(*Gestion des fronts demandes*)
FM_On.CLK	:=	CO_Etat;
FM_On();
IF FM_On.Q THEN
	VAR_Mem_CO_On	:=	TRUE;
END_IF
FD_Off.CLK	:=	CO_Etat;
FD_Off();
IF FD_Off.Q THEN
	VAR_Mem_CO_Off	:=	TRUE;
END_IF
FM_Regen.CLK	:=	CO_Regen;
FM_Regen();
IF FM_Regen.Q THEN
	VAR_Mem_CO_Regen	:=	TRUE;
	VAR_Mem_etape_Regen := TRUE;
END_IF
FM_states_regen.CLK	:=	CO_states_regen;
FM_states_regen();
IF FM_states_regen.Q THEN
	VAR_Mem_etape_Regen := TRUE;
END_IF
FM_StopRegen.CLK	:=	CO_StopRegen;
FM_StopRegen();
IF FM_StopRegen.Q THEN
	VAR_Mem_CO_StopRegen	:=	TRUE;
	VAR_Mem_etape_Regen := FALSE;
END_IF
FM_Param.CLK	:=	CO_Param_ParDefaut;
FM_Param();
IF FM_Param.Q THEN
	VAR_Mem_CO_Param_ParDefaut	:=	TRUE;
END_IF           
FM_Ecriture.CLK	:=	CO_Ecriture;
FM_Ecriture();
IF FM_Ecriture.Q THEN
	VAR_Mem_CO_Ecriture	:=	TRUE;
END_IF
FM_Lecture.CLK	:=	CO_Lecture;
FM_Lecture();
IF FM_Lecture.Q THEN
	VAR_Mem_CO_Lecture	:=	TRUE;
END_IF
FM_RoughValveOn.CLK	:=	CO_RoughValve;
FM_RoughValveOn();
IF FM_RoughValveOn.Q THEN
	VAR_Mem_CO_RoughValve_On	:=	TRUE;
END_IF
FM_PurgeValveOn.CLK	:=	CO_PurgeValve;
FM_PurgeValveOn();
IF FM_PurgeValveOn.Q THEN
	VAR_Mem_CO_PurgeValve_On	:=	TRUE;
END_IF
FM_RoughValveOff.CLK	:=	CO_RoughValve;
FM_RoughValveOff();
IF FM_RoughValveOff.Q THEN
	VAR_Mem_CO_RoughValve_Off	:=	TRUE;
END_IF
FM_PurgeValveOff.CLK	:=	CO_PurgeValve;
FM_PurgeValveOff();
IF FM_PurgeValveOff.Q THEN
	VAR_Mem_CO_PurgeValve_Off	:=	TRUE;
END_IF

FM_pump_TC_ON.CLK	:=	CO_PumpTc;
FM_pump_TC_ON();
IF FM_pump_TC_ON.Q THEN
	VAR_Mem_CO_PumpTC_on	:=	TRUE;
END_IF
FM_pump_TC_OFF.CLK	:=	CO_PumpTc;
FM_pump_TC_OFF();
IF FM_pump_TC_OFF.Q THEN
	VAR_Mem_CO_PumpTC_off	:=	TRUE;
END_IF



FM_InfoPompe.CLK	:=	CO_InfoPompe;
FM_InfoPompe();
IF FM_InfoPompe.Q THEN
	VAR_Mem_CO_Info_Pompe	:=	TRUE;
END_IF
FM_LectureRelay.CLK := CO_Lecture_Relay;
FM_LectureRelay();
IF FM_LectureRelay.Q THEN
	VAR_Mem_CO_Lecture_Relay:=TRUE;
END_IF
FM_EnvoieParamRelay.CLK	:=	CO_Envoie_Param_Relay;
FM_EnvoieParamRelay();
IF FM_EnvoieParamRelay.Q THEN
	VAR_Mem_CO_Envoie_Param_Relay	:=	TRUE;
END_IF
FM_ParamUsineRelay.CLK	:=	CO_Param_usine_Relay;
FM_ParamUsineRelay();
IF FM_ParamUsineRelay.Q THEN
	VAR_Mem_CO_Param_usine_Relay	:=	TRUE;
END_IF

IF NOT CO_Etat THEN
	STATE_Pompe:= FALSE;
END_IF

A_error:= OUT_Send_Data.Error;


(*RESET ou DESACTIVATION Driver*)
IF RESET OR OFF THEN
	VAR_Cadence                 := 0;
	STATE_Temperature[0]		:=	0;
	STATE_Temperature[1]		:=	0;
	STATE_Pressure        		:=  0;
	REGEN_ERROR                 := '';
	Reponse_ModeManu            := '';
	STEP_Regen                  := '';
	STATE_ROR_nb                := 0;
	LAST_ROR_Value              := 0;
	STATE_Rough_valve           := FALSE;
	STATE_Purge_valve           := FALSE;
	STEP_REGEN_ID               := 1000;
	VAR_Affichage               := '';
	Pump_Serial_Number_affiche	:= '';
	Number_Of_Complete_Regen    := 0;
	Time_Since_Last_Regen       := 0;
	SoftwareRevisionLevel       := '';
	ElaspedTime                 := 0;
	STATE_Tps_restant           := 0;
	VAR_Mem_CO_Ecriture   		:= FALSE;
	VAR_Mem_CO_Param_ParDefaut  := FALSE;
	VAR_Mem_CO_On				:= FALSE;
	VAR_Mem_CO_Off		  		:= TRUE ;
	VAR_Mem_CO_Regen	 		:= FALSE;
	VAR_Mem_CO_StopRegen 		:= TRUE ;
	VAR_Mem_CO_PurgeValve_off   := TRUE ;
	VAR_Mem_CO_PurgeValve_on    := FALSE;
	VAR_Mem_CO_RoughValve_off   := TRUE ;
	VAR_Mem_CO_RoughValve_on    := FALSE;
	VAR_Mem_CO_Info_Pompe		:= FALSE;
	RETURN;
END_IF



TIMER_Demarrage.IN 	:= 	NOT IN_Receive_Data.Busy AND NOT OUT_Send_Data.Busy AND NOT VAR_ReceptionOk;
TIMER_Demarrage.PT	:=	T#5S;
TIMER_Demarrage();
IF TIMER_Demarrage.Q  THEN
	VAR_ReceptionOk	:=	TRUE;
	VAR_Cadence 	:= 	1;
END_IF

(*Cadencement des trames*)
TIMER_Cadence(IN:=VAR_ReceptionOk, PT:=T#500MS);
VAR_Mem_Cadence	:=	VAR_Cadence;



(*GESTION ENVOI*)
IF TIMER_Cadence.Q AND NOT OUT_Send_Data.Busy AND NOT CO_ModeManu THEN
	VAR_STR2 := CHR(36);	(*$ = hex 24 = dec 36*)

	(* Remplissage trame : $ + code + checksum + 0D*)
	CASE VAR_Cadence OF

			1: 	(* Demande état on/off pompe*)
				VAR_BuffString		:= 	'';
				VAR_BuffString		:=	VAR_STR2;
				VAR_BuffString		:=	CONCAT(VAR_BuffString, 'A?');
				VAR_BuffString		:=	CONCAT(VAR_BuffString,CHECKSUM(VAR_BuffString,TRUE));
				VAR_BuffString		:=	CONCAT(VAR_BuffString,'$0D');
				OUT_Send_Data.SendString		:=	VAR_BuffString;

			2: 	(* Demande état regen pompe*)
				VAR_BuffString		:= 	'';
				VAR_BuffString		:=	VAR_STR2;
				VAR_BuffString		:=	CONCAT(VAR_BuffString, 'O');
				VAR_BuffString		:=	CONCAT(VAR_BuffString,CHECKSUM(VAR_BuffString,TRUE));
				VAR_BuffString		:=	CONCAT(VAR_BuffString,'$0D');
				OUT_Send_Data.SendString		:=	VAR_BuffString;
				
			3:	(* Demande erreur regen *)
				VAR_BuffString		:= 	'';
				VAR_BuffString		:=	VAR_STR2;
				VAR_BuffString		:=	CONCAT(VAR_BuffString, 'e');
				VAR_BuffString		:=	CONCAT(VAR_BuffString,CHECKSUM(VAR_BuffString,TRUE));
				VAR_BuffString		:=	CONCAT(VAR_BuffString,'$0D');
				OUT_Send_Data.SendString		:=	VAR_BuffString;
				
			4: 	(* Demande etat rough valve *)
				VAR_BuffString		:= 	'';
				VAR_BuffString		:=	VAR_STR2;
				VAR_BuffString		:=	CONCAT(VAR_BuffString, 'D?');
				VAR_BuffString		:=	CONCAT(VAR_BuffString,CHECKSUM(VAR_BuffString,TRUE));
				VAR_BuffString		:=	CONCAT(VAR_BuffString,'$0D');
				OUT_Send_Data.SendString	:=	VAR_BuffString;
				
			5: 	(* Demande etat purge valve *)
				VAR_BuffString		:= 	'';
				VAR_BuffString		:=	VAR_STR2;
				VAR_BuffString		:=	CONCAT(VAR_BuffString, 'E?');
				VAR_BuffString		:=	CONCAT(VAR_BuffString,CHECKSUM(VAR_BuffString,TRUE));
				VAR_BuffString		:=	CONCAT(VAR_BuffString,'$0D');
				OUT_Send_Data.SendString	:=	VAR_BuffString;
		
			
			6: 	(* Demande température étage 1*)
				VAR_BuffString		:= 	'';
				VAR_BuffString		:=	VAR_STR2;
				VAR_BuffString		:=	CONCAT(VAR_BuffString, 'J');
				VAR_BuffString		:=	CONCAT(VAR_BuffString,CHECKSUM(VAR_BuffString,TRUE));
				VAR_BuffString		:=	CONCAT(VAR_BuffString,CHR(13));
				VAR_TrameRetour     :=  VAR_BuffString;
				OUT_Send_Data.SendString	:=	VAR_BuffString;
				
			7: 	(* Demande température étage 2*)
				VAR_BuffString		:= 	'';
				VAR_BuffString		:=	VAR_STR2;
				VAR_BuffString		:=	CONCAT(VAR_BuffString, 'K');
				VAR_BuffString		:=	CONCAT(VAR_BuffString,CHECKSUM(VAR_BuffString,TRUE));
				VAR_BuffString		:=	CONCAT(VAR_BuffString,'$0D');
				OUT_Send_Data.SendString		:=	VAR_BuffString;
				
			8: 	(* Demande pression *)
				VAR_BuffString		:= 	'';
				VAR_BuffString		:=	VAR_STR2;
				VAR_BuffString		:=	CONCAT(VAR_BuffString, 'L');
				VAR_BuffString		:=	CONCAT(VAR_BuffString,CHECKSUM(VAR_BuffString,TRUE));
				VAR_BuffString		:=	CONCAT(VAR_BuffString,'$0D');
				OUT_Send_Data.SendString	:=	VAR_BuffString;
				
			9: 	(* Demande etat pump TC *)
				VAR_BuffString		:= 	'';
				VAR_BuffString		:=	VAR_STR2;
				VAR_BuffString		:=	CONCAT(VAR_BuffString, 'B?');
				VAR_BuffString		:=	CONCAT(VAR_BuffString,CHECKSUM(VAR_BuffString,TRUE));
				VAR_BuffString		:=	CONCAT(VAR_BuffString,'$0D');
				OUT_Send_Data.SendString	:=	VAR_BuffString;	
		
			10:	(* Demande de regen/arret regen d'une pompe *)
				VAR_BuffString		:= 	'';
				VAR_BuffString		:=	VAR_STR2;
				IF VAR_Mem_CO_Regen AND NOT VAR_Mem_CO_StopRegen THEN
					VAR_BuffString		:=	CONCAT(VAR_BuffString,'N1');
				ELSIF VAR_Mem_CO_StopRegen THEN
					VAR_BuffString		:=	CONCAT(VAR_BuffString,'N0');
				END_IF
				VAR_BuffString		:=	CONCAT(VAR_BuffString,CHECKSUM(VAR_BuffString,TRUE));
				VAR_BuffString		:=	CONCAT(VAR_BuffString,'$0D');
				OUT_Send_Data.SendString		:=	VAR_BuffString;
				
			11: 	(* Demande de marche ou d'arrêt d'une pompe *)
				VAR_BuffString		:= 	'';
				VAR_BuffString		:=	VAR_STR2;
				IF	CO_ETAT THEN
					VAR_BuffString	:=	CONCAT(VAR_BuffString,'A1');
				ELSE
					VAR_BuffString	:=	CONCAT(VAR_BuffString,'A0');
				END_IF
				VAR_BuffString		:=	CONCAT(VAR_BuffString,CHECKSUM(VAR_BuffString,TRUE));
				VAR_BuffString		:=	CONCAT(VAR_BuffString,'$0D');
				OUT_Send_Data.SendString		:=	VAR_BuffString;
				
			12:  (*paramètre de la regen en ecriture*)
				PRM_PowerFailRecovery:= ID_COMBOBOX;
				IF VAR_Mem_CO_Ecriture AND VAR_Reception_Parametre THEN
				VAR_BuffString	:= 	'';
				VAR_BuffString	:=	VAR_STR2;
				CASE iCounter_Regen_ecriture OF 
					0:	
						VAR_BuffString	:=	CONCAT(VAR_BuffString,'P');
						VAR_BuffString	:=	CONCAT(VAR_BuffString,INT_TO_STRING(iCounter_Regen_ecriture));
						VAR_BuffString	:=	CONCAT(VAR_BuffString,UINT_TO_STRING(REAL_TO_UINT(LIMIT(0,60 * PRM_PumpRestartDelay,59994))));
					1:	
						VAR_BuffString	:=	CONCAT(VAR_BuffString,'P');
						VAR_BuffString	:=	CONCAT(VAR_BuffString,INT_TO_STRING(iCounter_Regen_ecriture));
						VAR_BuffString	:=	CONCAT(VAR_BuffString,UINT_TO_STRING(LIMIT(0,PRM_ExtendedPurgeTime,9999)));
					2:	
						VAR_BuffString	:=	CONCAT(VAR_BuffString,'P');
						VAR_BuffString	:=	CONCAT(VAR_BuffString,INT_TO_STRING(iCounter_Regen_ecriture));
						VAR_BuffString	:=	CONCAT(VAR_BuffString,UINT_TO_STRING(LIMIT(0,PRM_RepurgeCycles,20)));
					3:
						VAR_BuffString	:=	CONCAT(VAR_BuffString,'P');
					   	VAR_BuffString	:=	CONCAT(VAR_BuffString,INT_TO_STRING(iCounter_Regen_ecriture));
						VAR_BuffString	:=	CONCAT(VAR_BuffString,UINT_TO_STRING(LIMIT(25,PRM_RoughToPressure,200)));
					4:	
						VAR_BuffString	:=	CONCAT(VAR_BuffString,'P');
						VAR_BuffString	:=	CONCAT(VAR_BuffString,INT_TO_STRING(iCounter_Regen_ecriture));
						VAR_BuffString	:=	CONCAT(VAR_BuffString,UINT_TO_STRING(LIMIT(1,PRM_ROR,100)));
					5:	
						VAR_BuffString	:=	CONCAT(VAR_BuffString,'P');
						VAR_BuffString	:=	CONCAT(VAR_BuffString,INT_TO_STRING(iCounter_Regen_ecriture));
						VAR_BuffString	:=	CONCAT(VAR_BuffString,UINT_TO_STRING(LIMIT(0,PRM_RORCycles,40)));
					6:	
						VAR_BuffString	:=	CONCAT(VAR_BuffString,'P');
						VAR_BuffString	:=	CONCAT(VAR_BuffString,INT_TO_STRING(iCounter_Regen_ecriture));
						VAR_BuffString	:=	CONCAT(VAR_BuffString,UINT_TO_STRING(LIMIT(10,PRM_StartUpTemperature,80)));
					7:	
						VAR_BuffString	:=	CONCAT(VAR_BuffString,'P');
						VAR_BuffString	:=	CONCAT(VAR_BuffString,'A');
						VAR_BuffString	:=	CONCAT(VAR_BuffString,INT_TO_STRING(BOOL_TO_INT(PRM_RoughValveInterlock)));
					8:	
						VAR_BuffString	:=	CONCAT(VAR_BuffString,'P');
						VAR_BuffString	:=	CONCAT(VAR_BuffString,'G');
						VAR_BuffString	:=	CONCAT(VAR_BuffString,REAL_TO_STRING(LIMIT(0,PRM_RepurgeTime,9999)));
					9:
						VAR_BuffString	:=	CONCAT(VAR_BuffString,'j');
						VAR_BuffString	:=	CONCAT(VAR_BuffString,UINT_TO_STRING(REAL_TO_UINT(LIMIT(0,60*PRM_PumpStartDelay,9999))));
					10:
						VAR_BuffString	:=	CONCAT(VAR_BuffString,'i');
						VAR_BuffString	:=	CONCAT(VAR_BuffString,USINT_TO_STRING(LIMIT(0,PRM_PowerFailRecovery,2)));
					11:    
						VAR_BuffString	:=	CONCAT(VAR_BuffString,'H');
						VAR_BuffString	:=	CONCAT(VAR_BuffString,UINT_TO_STRING(LIMIT(0,PRM_1st_stage_control_temp,320)));    
				END_CASE
				VAR_BuffString		:=	CONCAT(VAR_BuffString,CHECKSUM(VAR_BuffString,TRUE));
				VAR_BuffString		:=	CONCAT(VAR_BuffString,'$0D');
				iCounter_Regen_ecriture := iCounter_Regen_ecriture + 1;
				OUT_Send_Data.SendString := VAR_BuffString;
				IF iCounter_Regen_ecriture >=12 THEN
					iCounter_Regen_ecriture := 0;
				END_IF
				VAR_Reception_Parametre := FALSE;	
				END_IF
			13:(*paramètre de la regen en lecture*)
				IF VAR_Mem_CO_Lecture AND VAR_Reception_Parametre THEN
				VAR_BuffString		:= 	'';
				VAR_BuffString		:=	VAR_STR2;
				
				CASE iCounter_Regen_lecture OF 
					0:
						VAR_BuffString	:=	CONCAT(VAR_BuffString,'i');
					1:	
						VAR_BuffString	:=	CONCAT(VAR_BuffString,'P');
						VAR_BuffString	:=	CONCAT(VAR_BuffString,'6');
					2:
						VAR_BuffString	:=	CONCAT(VAR_BuffString,'j');
					3:
						VAR_BuffString	:=	CONCAT(VAR_BuffString,'P');
						VAR_BuffString	:=	CONCAT(VAR_BuffString,INT_TO_STRING(0));
					4:
						VAR_BuffString	:=	CONCAT(VAR_BuffString,'P');
						VAR_BuffString	:=	CONCAT(VAR_BuffString,INT_TO_STRING(1));
					5:	
						VAR_BuffString	:=	CONCAT(VAR_BuffString,'P');
						VAR_BuffString	:=	CONCAT(VAR_BuffString,INT_TO_STRING(2));
					6:	
						VAR_BuffString	:=	CONCAT(VAR_BuffString,'P');
						VAR_BuffString	:=	CONCAT(VAR_BuffString,'G');
					7:	
						VAR_BuffString	:=	CONCAT(VAR_BuffString,'P');
					    VAR_BuffString	:=	CONCAT(VAR_BuffString,INT_TO_STRING(4));
					8:	
						VAR_BuffString	:=	CONCAT(VAR_BuffString,'P');
						VAR_BuffString	:=	CONCAT(VAR_BuffString,INT_TO_STRING(5));
					9:	
						VAR_BuffString	:=	CONCAT(VAR_BuffString,'P');
						VAR_BuffString	:=	CONCAT(VAR_BuffString,INT_TO_STRING(3));
					10:
						VAR_BuffString	:=	CONCAT(VAR_BuffString,'P');
						VAR_BuffString	:=	CONCAT(VAR_BuffString,'A');
					11:
						VAR_BuffString	:=	CONCAT(VAR_BuffString,'H');
				END_CASE
				VAR_BuffString	:=	CONCAT(VAR_BuffString,'?');
				VAR_BuffString	:=	CONCAT(VAR_BuffString,CHECKSUM(VAR_BuffString,TRUE));
				VAR_BuffString	:=	CONCAT(VAR_BuffString,'$0D');
				
				OUT_Send_Data.SendString  :=	VAR_BuffString;
				VAR_Reception_Parametre := FALSE;
				END_IF	
				
			14: (* lecture des informations de la regen *)
				CASE iCounter_Valeur_Num_Regen OF 
					0:	
						VAR_BuffString		:= 	'';
						VAR_BuffString		:=	VAR_STR2;
						VAR_BuffString		:=	CONCAT(VAR_BuffString,'O');
						VAR_BuffString		:=	CONCAT(VAR_BuffString,CHECKSUM(VAR_BuffString,TRUE));
						VAR_BuffString		:=	CONCAT(VAR_BuffString,'$0D');
						OUT_Send_Data.SendString :=	VAR_BuffString;
						
					1:
						VAR_BuffString		:= 	'';
						VAR_BuffString		:=	VAR_STR2;
						VAR_BuffString		:=	CONCAT(VAR_BuffString, 'K');
						VAR_BuffString		:=	CONCAT(VAR_BuffString,CHECKSUM(VAR_BuffString,TRUE));
						VAR_BuffString		:=	CONCAT(VAR_BuffString,'$0D');
						OUT_Send_Data.SendString		:=	VAR_BuffString;
						
					2:
						VAR_BuffString		:= 	'';
						VAR_BuffString		:=	VAR_STR2;
						VAR_BuffString		:=	CONCAT(VAR_BuffString, 'L');
						VAR_BuffString		:=	CONCAT(VAR_BuffString,CHECKSUM(VAR_BuffString,TRUE));
						VAR_BuffString		:=	CONCAT(VAR_BuffString,'$0D');
						OUT_Send_Data.SendString		:=	VAR_BuffString;
					
					3: 
						VAR_BuffString		:= 	'';
						VAR_BuffString		:=	VAR_STR2;
						VAR_BuffString		:=	CONCAT(VAR_BuffString, 'e');
						VAR_BuffString		:=	CONCAT(VAR_BuffString,CHECKSUM(VAR_BuffString,TRUE));
						VAR_BuffString		:=	CONCAT(VAR_BuffString,'$0D');
						OUT_Send_Data.SendString		:=	VAR_BuffString;
						
					4:
						VAR_BuffString		:= 	'';
						VAR_BuffString		:=	VAR_STR2;
						VAR_BuffString		:=	CONCAT(VAR_BuffString, 'k');
						VAR_BuffString		:=	CONCAT(VAR_BuffString,CHECKSUM(VAR_BuffString,TRUE));
						VAR_BuffString		:=	CONCAT(VAR_BuffString,'$0D');
						OUT_Send_Data.SendString		:=	VAR_BuffString;
						
					5:
						VAR_BuffString		:= 	'';
						VAR_BuffString		:=	VAR_STR2;
						VAR_BuffString		:=	CONCAT(VAR_BuffString, 'm');
						VAR_BuffString		:=	CONCAT(VAR_BuffString,CHECKSUM(VAR_BuffString,TRUE));
						VAR_BuffString		:=	CONCAT(VAR_BuffString,'$0D');
						OUT_Send_Data.SendString		:=	VAR_BuffString;
					
					6:
						VAR_BuffString		:= 	'';
						VAR_BuffString		:=	VAR_STR2;
						VAR_BuffString		:=	CONCAT(VAR_BuffString, 'n');
						VAR_BuffString		:=	CONCAT(VAR_BuffString,CHECKSUM(VAR_BuffString,TRUE));
						VAR_BuffString		:=	CONCAT(VAR_BuffString,'$0D');
						OUT_Send_Data.SendString		:=	VAR_BuffString;
						
					7:
						VAR_BuffString		:= 	'';
						VAR_BuffString		:=	VAR_STR2;
						VAR_BuffString		:=	CONCAT(VAR_BuffString, 'A?');
						VAR_BuffString		:=	CONCAT(VAR_BuffString,CHECKSUM(VAR_BuffString,TRUE));
						VAR_BuffString		:=	CONCAT(VAR_BuffString,'$0D');
						OUT_Send_Data.SendString		:=	VAR_BuffString;
						
					8: 	(* Demande rough valve *)
						VAR_BuffString		:= 	'';
						VAR_BuffString		:=	VAR_STR2;
						VAR_BuffString		:=	CONCAT(VAR_BuffString, 'D?');
						VAR_BuffString		:=	CONCAT(VAR_BuffString,CHECKSUM(VAR_BuffString,TRUE));
						VAR_BuffString		:=	CONCAT(VAR_BuffString,'$0D');
						OUT_Send_Data.SendString	:=	VAR_BuffString;
				
					9: 	(* Demande purge valve *)
						VAR_BuffString		:= 	'';
						VAR_BuffString		:=	VAR_STR2;
						VAR_BuffString		:=	CONCAT(VAR_BuffString, 'E?');
						VAR_BuffString		:=	CONCAT(VAR_BuffString,CHECKSUM(VAR_BuffString,TRUE));
						VAR_BuffString		:=	CONCAT(VAR_BuffString,'$0D');
						OUT_Send_Data.SendString	:=	VAR_BuffString;
						
					10: (*demande nombre de cycle de purge fail*)
						VAR_BuffString		:= 	'';
						VAR_BuffString		:=	VAR_STR2;
						VAR_BuffString		:=	CONCAT(VAR_BuffString, 'l');
						VAR_BuffString		:=	CONCAT(VAR_BuffString,CHECKSUM(VAR_BuffString,TRUE));
						VAR_BuffString		:=	CONCAT(VAR_BuffString,'$0D');
						OUT_Send_Data.SendString		:=	VAR_BuffString;
					11:	
						VAR_BuffString		:= 	'';
						VAR_BuffString		:=	VAR_STR2;
						VAR_BuffString		:=	CONCAT(VAR_BuffString, 'J');
						VAR_BuffString		:=	CONCAT(VAR_BuffString,CHECKSUM(VAR_BuffString,TRUE));
						VAR_BuffString		:=	CONCAT(VAR_BuffString,'$0D');
						OUT_Send_Data.SendString		:=	VAR_BuffString;
				END_CASE
				
					15:	(* Demande de ouverture/fermeture rough valve *)
						VAR_BuffString		:= 	'';
						VAR_BuffString		:=	VAR_STR2;
						IF CO_RoughValve THEN
							VAR_BuffString		:=	CONCAT(VAR_BuffString,'D1');
						ELSIF NOT CO_RoughValve THEN
							VAR_BuffString		:=	CONCAT(VAR_BuffString,'D0');
						END_IF
						VAR_BuffString		:=	CONCAT(VAR_BuffString,CHECKSUM(VAR_BuffString,TRUE));
						VAR_BuffString		:=	CONCAT(VAR_BuffString,'$0D');
						OUT_Send_Data.SendString		:=	VAR_BuffString;
					
					16:	(* Demande de ouverture/fermeture purge valve *)
						VAR_BuffString		:= 	'';
						VAR_BuffString		:=	VAR_STR2;
						IF CO_PurgeValve THEN
							VAR_BuffString		:=	CONCAT(VAR_BuffString,'E1');
						ELSIF NOT CO_PurgeValve THEN
							VAR_BuffString		:=	CONCAT(VAR_BuffString,'E0');
						END_IF
						VAR_BuffString		:=	CONCAT(VAR_BuffString,CHECKSUM(VAR_BuffString,TRUE));
						VAR_BuffString		:=	CONCAT(VAR_BuffString,'$0D');
						OUT_Send_Data.SendString		:=	VAR_BuffString;
						
					17: (* informations supplémentaire pompe*)
						VAR_BuffString		:= 	'';
						VAR_BuffString		:=	VAR_STR2;
						CASE iCounter_Info_Pompe OF 
							0:
								VAR_BuffString		:=	CONCAT(VAR_BuffString,'VA?');		(*premiere parti du num de serie*)
							1:
								VAR_BuffString		:=	CONCAT(VAR_BuffString,'VQ?');		(*deuxième parti du num de serie*)
							2:
								VAR_BuffString		:=	CONCAT(VAR_BuffString,'Z?');		(*nb de regen complete*)
							3:
								VAR_BuffString		:=	CONCAT(VAR_BuffString,'a');			(*tps depuis la dernière regen*)
							4:
								VAR_BuffString		:=	CONCAT(VAR_BuffString,'@');			(*version logiciel*)	
							5:
								VAR_BuffString		:=	CONCAT(VAR_BuffString,'Y?');		(*tps de fonctionnement de la pompe*)
						END_CASE
						VAR_BuffString		:=	CONCAT(VAR_BuffString,CHECKSUM(VAR_BuffString,TRUE));
						VAR_BuffString		:=	CONCAT(VAR_BuffString,'$0D');
						OUT_Send_Data.SendString		:=	VAR_BuffString;
						
					18:
						(*envoie param relay*)
						VAR_BuffString		:= 	'';
						VAR_BuffString		:=	VAR_STR2;
						var_STRING :=	BYTE_TO_HEXSTR(USINT_TO_BYTE(PRM_Action),1,FALSE);
								IF PRM_Mode THEN
									VAR_BuffString		:=	CONCAT(VAR_BuffString,'[B' );
									VAR_BuffString      :=  CONCAT(VAR_BuffString,USINT_TO_STRING(PRM_Relay));
								ELSIF PRM_Mode=FALSE THEN
									IF PRM_Action =10 OR PRM_Action =11 OR PRM_Action =12 OR PRM_Action =13 OR PRM_Action =15 THEN
										VAR_BuffString		:=	CONCAT(VAR_BuffString,'T' );
										VAR_BuffString      :=  CONCAT(VAR_BuffString,USINT_TO_STRING(PRM_Relay));
										VAR_BuffString		:=	CONCAT(VAR_BuffString,BYTE_TO_HEXSTR(USINT_TO_BYTE(PRM_Action),1,FALSE));
									ELSE
										VAR_BuffString		:=	CONCAT(VAR_BuffString,'T' );
										VAR_BuffString      :=  CONCAT(VAR_BuffString,USINT_TO_STRING(PRM_Relay));
										VAR_BuffString		:=	CONCAT(VAR_BuffString,BYTE_TO_HEXSTR(USINT_TO_BYTE(PRM_Action),1,FALSE));
										IF PRM_Action=0 THEN
											VAR_BuffString	:=	CONCAT(VAR_BuffString,UINT_TO_STRING(LIMIT(30,PRM_Valeur,310)));
										ELSIF PRM_Action=1 THEN
											VAR_BuffString	:=	CONCAT(VAR_BuffString,UINT_TO_STRING(LIMIT(30,PRM_Valeur,310)));
										ELSIF PRM_Action=2 THEN
											VAR_BuffString	:=	CONCAT(VAR_BuffString,UINT_TO_STRING(LIMIT(10,PRM_Valeur,310)));
										ELSIF PRM_Action=3 THEN
											VAR_BuffString	:=	CONCAT(VAR_BuffString,UINT_TO_STRING(LIMIT(10,PRM_Valeur,310)));
										ELSIF PRM_Action=4 THEN
											VAR_BuffString	:=	CONCAT(VAR_BuffString,UINT_TO_STRING(LIMIT(1,PRM_Valeur,999)));
										ELSIF PRM_Action=5 THEN
											VAR_BuffString	:=	CONCAT(VAR_BuffString,UINT_TO_STRING(LIMIT(1,PRM_Valeur,999)));
										ELSIF PRM_Action=6 THEN
											VAR_BuffString	:=	CONCAT(VAR_BuffString,UINT_TO_STRING(LIMIT(1,PRM_Valeur,999)));
										ELSIF PRM_Action=7 THEN
											VAR_BuffString	:=	CONCAT(VAR_BuffString,UINT_TO_STRING(LIMIT(1,PRM_Valeur,999)));
										ELSIF PRM_Action=8 THEN
											VAR_BuffString	:=	CONCAT(VAR_BuffString,UINT_TO_STRING(LIMIT(0,PRM_Valeur,9999)));
										END_IF	
									END_IF
								END_IF
						VAR_BuffString		:=	CONCAT(VAR_BuffString,CHECKSUM(VAR_BuffString,TRUE));
						VAR_BuffString		:=	CONCAT(VAR_BuffString,'$0D');
						OUT_Send_Data.SendString		:=	VAR_BuffString;
						Var_lancement_timer_ONOFF := TRUE;
					19:
						(* lecture des parametres des relais*)
						VAR_BuffString		:= 	'';
						VAR_BuffString		:=	VAR_STR2;
						VAR_BuffString		:=	CONCAT(VAR_BuffString,'T' );
						VAR_BuffString		:=	CONCAT(VAR_BuffString, USINT_TO_STRING(PRM_Relay));
						VAR_BuffString		:=	CONCAT(VAR_BuffString, '?');
						CASE iCounter_Param_Relay_lecture OF 
							0:
								VAR_BuffString		:=	CONCAT(VAR_BuffString, '2');
							1:
								VAR_BuffString		:=	CONCAT(VAR_BuffString, '0');
							2: 
								VAR_BuffString		:=	CONCAT(VAR_BuffString, '1');             
							3:
								VAR_BuffString		:=	CONCAT(VAR_BuffString,'8');
						END_CASE
						VAR_BuffString		:=	CONCAT(VAR_BuffString,CHECKSUM(VAR_BuffString,TRUE));
						VAR_BuffString		:=	CONCAT(VAR_BuffString,'$0D');
						OUT_Send_Data.SendString		:=	VAR_BuffString;
					20:
						VAR_BuffString		:= 	'';
						VAR_BuffString		:=	VAR_STR2;
						CASE iCounter_Param_ParDefaut_Relay_lecture OF 
							0:
								VAR_BuffString		:=	CONCAT(VAR_BuffString,'T' );	
								VAR_BuffString		:=	CONCAT(VAR_BuffString, '1');	//relai
								VAR_BuffString		:=	CONCAT(VAR_BuffString, 'C');	//commande
							1:
								VAR_BuffString		:=	CONCAT(VAR_BuffString,'T' );
								VAR_BuffString		:=	CONCAT(VAR_BuffString, '2');	 //relai
								VAR_BuffString		:=	CONCAT(VAR_BuffString, '2');     //commande
								VAR_BuffString		:=	CONCAT(VAR_BuffString, '15');    //valeur
							2:
								VAR_BuffString		:=	CONCAT(VAR_BuffString,'T' );
								VAR_BuffString		:=	CONCAT(VAR_BuffString, '2');	 //relai
								VAR_BuffString		:=	CONCAT(VAR_BuffString, '3');	 //commande
								VAR_BuffString		:=	CONCAT(VAR_BuffString, '25');    //valeur
						END_CASE
						VAR_BuffString		:=	CONCAT(VAR_BuffString,CHECKSUM(VAR_BuffString,TRUE));
						VAR_BuffString		:=	CONCAT(VAR_BuffString,'$0D');
						OUT_Send_Data.SendString		:=	VAR_BuffString;
						
					21:	(* Demande de ouverture/fermeture rough valve *)
						VAR_BuffString		:= 	'';
						VAR_BuffString		:=	VAR_STR2;
						IF CO_PumpTc THEN
							VAR_BuffString		:=	CONCAT(VAR_BuffString,'B1');
						ELSIF NOT CO_PumpTc THEN
							VAR_BuffString		:=	CONCAT(VAR_BuffString,'B0');
						END_IF
						VAR_BuffString		:=	CONCAT(VAR_BuffString,CHECKSUM(VAR_BuffString,TRUE));
						VAR_BuffString		:=	CONCAT(VAR_BuffString,'$0D');
						OUT_Send_Data.SendString		:=	VAR_BuffString;
	END_CASE	
	

	(*Envoi*)
	OUT_Send_Data(TXbuffer:= OUT_Buffer);

	(* Reset timer *)
	VAR_ReceptionOk := FALSE;
ELSE
	IF CO_ModeManu AND CO_EnvoiManu THEN
		OUT_Send_Data.SendString	:=	VAR_BuffString;
		(*Envoi*)
		OUT_Send_Data(TXbuffer:= OUT_Buffer);
		CO_EnvoiManu		:=	FALSE;
		VAR_ReceptionOk 	:= 	FALSE;
	END_IF
END_IF

IF VAR_Mem_CO_Param_ParDefaut THEN 					(*paramètre de regen par defaut + envoie*)
	PRM_PumpRestartDelay :=	0;                   
	ID_COMBOBOX := 1;
	PRM_ExtendedPurgeTime := 60;
	PRM_RepurgeCycles:=  10;
	PRM_RoughToPressure := 80;
	PRM_ROR := 16;
	PRM_RORCycles := 20;
	PRM_StartUpTemperature := 45;
	PRM_RoughValveInterlock := 0;
	PRM_RepurgeTime := 10;
	PRM_PumpStartDelay := 0.1;
	VAR_Mem_CO_Ecriture:= TRUE;
	VAR_Mem_CO_Param_ParDefaut:=FALSE;
END_IF
IF CO_ModeManu THEN               (*trame mode manu*)
		VAR_STR1 		:= 	CHECKSUM(PRM_TrameManu ,FALSE);
		VAR_STR2		:=	chr(36);
		VAR_BuffString	:=	CONCAT(VAR_STR2,PRM_TrameManu);
		VAR_BuffString	:=	CONCAT(VAR_BuffString,VAR_STR1);
		VAR_BuffString	:=	CONCAT(VAR_BuffString,CHR(13));
END_IF

(*GESTION RECEPTION*)
(*Réception*)
IN_Receive_Data(
	(*Prefix := chr(36),*)
	Suffix:= chr(13),
	Timeout:= T#1S,
	Reset :=OFF,
	ReceivedString := VAR_TrameRetour,
	RXbuffer := IN_Buffer);
 
	
(*interprétation trame retour*)
IF IN_Receive_Data.StringReceived THEN
	IF NOT CO_ModeManu THEN
		CASE VAR_Cadence OF

			1: (* Demande état On/off pompe *)
				VAR_STR1	:=	MID(VAR_TrameRetour,1,3);
				STATE_Pompe	:=	(VAR_STR1 = '1');

			2: (* Demande état regen pompe *)
				VAR_STR1	:=	MID(VAR_TrameRetour,1,3);
				STATE_Regen	:=	NOT((VAR_STR1 = 'V') OR (VAR_STR1 = 'P'));
				IF (VAR_STR1 = 'P') THEN
					STEP_Regen := 'REGEN COMPLETED';
					STEP_REGEN_ID := 34;
					Regen_completed:= TRUE;
				ELSIF (VAR_STR1 = 'V') THEN
					STEP_Regen := 'REGEN ABORTED';
					STEP_REGEN_ID := 35;
					Regen_completed:=FALSE;
				END_IF
				
			3:  (* Demande erreur regen *)
				VAR_STR1	:=	MID(VAR_TrameRetour,1,3);
				IF (VAR_STR1 = 'B') THEN 
							ID_ERREUR_REGEN := 58 ;
							REGEN_ERROR := 'WARMUP TIMEOUT';
				ELSIF (VAR_STR1 = '@')AND (CO_Regen = FALSE) THEN
							ID_ERREUR_REGEN := 59;
							REGEN_ERROR := 'NO ERROR'; 
				ELSIF (VAR_STR1 = 'C') THEN
							ID_ERREUR_REGEN := 60;
							REGEN_ERROR := 'COOLDOWN TIMEOUT';
				ELSIF (VAR_STR1 = 'D') THEN
							ID_ERREUR_REGEN := 61;
							REGEN_ERROR := 'ERROR IN ROR';
				ELSIF (VAR_STR1 = 'E') THEN
							ID_ERREUR_REGEN := 62;
							REGEN_ERROR := 'ROR CYCLE LIMIT WAS REACHED';
				ELSIF (VAR_STR1 = 'F') THEN 
							ID_ERREUR_REGEN := 63;
							//REGEN_ERROR := 'MANUAL ABORT';
				ELSIF (VAR_STR1 = 'G') THEN
							ID_ERREUR_REGEN := 64;
							REGEN_ERROR := 'ROUGH VALVE TIMEOUT';
				ELSIF (VAR_STR1 = 'H') THEN
					ID_ERREUR_REGEN := 65;
					REGEN_ERROR := 'system bug';
				ELSE
					ID_ERREUR_REGEN := 1000;
				END_IF
				VAR_Affichage1 := '';          						(*affichage de l'erreur, ce qui arreté la regen*)
				VAR_Affichage2 := '';       
				VAR_Affichage3 := '';
				VAR_Affichage:= CONCAT(VAR_Affichage1, VAR_Affichage2);
				VAR_Affichage:=CONCAT(VAR_Affichage, VAR_Affichage3);
				
			4: (* set rough valve*)
				VAR_STR1	:=	MID(VAR_TrameRetour,1,3);
				STATE_Rough_valve	:=	(VAR_STR1 = '1');
			
			5: (* set purge valve*)
				VAR_STR1	:=	MID(VAR_TrameRetour,1,3);
				STATE_Purge_valve	:=	(VAR_STR1 = '1');
				
			6: (* demande température étage 1*)
				STATE_Temperature[0]	:=	STRING_TO_REAL(MID(VAR_TrameRetour,6,4));

			7: (* demande température étage 2*)
				STATE_Temperature[1]	:=	STRING_TO_REAL(MID(VAR_TrameRetour,6,4));
				
			8: (* demande pression*)
				STATE_Pressure	:=	STRING_TO_REAL(MID(VAR_TrameRetour,6,4));
			
			9: (* set pump TC*)
				VAR_STR1	:=	MID(VAR_TrameRetour,1,3);
				STATE_Pump_TC	:=	(VAR_STR1 = '1');
				
			10: (* Demande de regen ou arrêt regen d'une pompe *)
				VAR_Mem_CO_StopRegen	:=	FALSE;
				VAR_Mem_CO_Regen	:=	FALSE;
				
				
			11: (* Demande de marche ou d'arrêt d'une pompe *)
				VAR_Mem_CO_Off	:=	FALSE;
				VAR_Mem_CO_On	:=	FALSE;
				
			12: (*ecriture parametre regen ecriture *)
				VAR_Reception_Parametre := TRUE;
				IF iCounter_Regen_ecriture = 0 THEN 
					VAR_Mem_CO_Ecriture := FALSE;
				END_IF
				
			13:  (* Demande lecture parametre regen pompe *)
				VAR_Reception_Parametre := TRUE;
				CASE iCounter_Regen_lecture OF 
					0:
						ID_COMBOBOX := STRING_TO_USINT(MID(VAR_TrameRetour,1,3));
						(*PRM_PowerFailRecovery_lecture := STRING_TO_USINT(MID(VAR_TrameRetour,1,3));*)
						PRM_PowerFailRecovery := STRING_TO_USINT(MID(VAR_TrameRetour,1,3));
					1: 
						PRM_StartUpTemperature := STRING_TO_USINT(MID(VAR_TrameRetour,2,8));
					2:
						PRM_PumpStartDelay := STRING_TO_REAL(MID(VAR_TrameRetour,4,4))/60;
					3: 
						PRM_PumpRestartDelay :=	STRING_TO_REAL(MID(VAR_TrameRetour,5,4))/60;                   (*ajouter la fonction lecture valeur*)
					4:
						PRM_ExtendedPurgeTime := STRING_TO_UINT(MID(VAR_TrameRetour,4,4));
					5:
						PRM_RepurgeCycles  := STRING_TO_USINT(MID(VAR_TrameRetour,2,4));
					6: 
						PRM_RepurgeTime := STRING_TO_USINT(MID(VAR_TrameRetour,4,4));
					7:
						PRM_ROR := STRING_TO_USINT(MID(VAR_TrameRetour,3,4));
					8:
						PRM_RORCycles := STRING_TO_USINT(MID(VAR_TrameRetour,2,4));
					9:
						PRM_RoughToPressure  :=	STRING_TO_USINT(MID(VAR_TrameRetour,3,4));
					10:
						PRM_RoughValveInterlock := STRING_TO_BOOL(MID(VAR_TrameRetour,1,3));
					11:
						PRM_1st_stage_control_temp := STRING_TO_USINT(MID(VAR_TrameRetour,6,4));
				END_CASE
				iCounter_Regen_lecture := iCounter_Regen_lecture + 1;
				IF iCounter_Regen_lecture >=12 THEN
					iCounter_Regen_lecture := 0;
					VAR_Mem_CO_lecture := FALSE;
					CO_Lecture:=FALSE;
				END_IF
				
		
						
			14:  (* Demande étape regen pompe + affichage numérique*)
				STATE_Regen:= NOT(VAR_STR1 = 'P' OR VAR_STR1 = 'V');
				CASE iCounter_Valeur_Num_Regen OF
					0:
						VAR_STR1	:=	MID(VAR_TrameRetour,1,3);
						IF (VAR_STR1 = 'A') OR (VAR_STR1 = '\')THEN 
							STEP_Regen := 'CRYO OFF';
							VAR_Affichage1 := '';          
							VAR_Affichage2 := '';       
							VAR_Affichage3 := '';
							STEP_REGEN_ID := 44 ;
							ID_ERREUR_REGEN := 1000;
							Regen_completed:=FALSE;
							VAR_Demande_Erreur:=FALSE;
						ELSIF (VAR_STR1 = 'B') OR (VAR_STR1 ='C')OR (VAR_STR1 = 'E') OR (VAR_STR1 ='Q') OR  (VAR_STR1 ='R') OR (VAR_STR1 ='^')  OR (VAR_STR1 =']') THEN 
							STEP_Regen := 'WARM-UP';
							VAR_Affichage1 := REAL_TO_STRING(STATE_Temperature[0]);          
							VAR_Affichage2 := '';       
							VAR_Affichage3 := '/310K';
							STEP_REGEN_ID := 26 ;
							ID_ERREUR_REGEN := 1001;
							Regen_completed:=FALSE;
							VAR_Demande_Erreur:=FALSE;
						ELSIF (VAR_STR1 = 'D') OR (VAR_STR1 ='F')OR (VAR_STR1 = 'G') THEN
							STEP_Regen := 'PURGE GAS FAILURE';
							STEP_REGEN_ID := 27 ;
							ID_ERREUR_REGEN := 1001;
							Regen_completed:=FALSE;
							VAR_Demande_Erreur:=FALSE;
						ELSIF (VAR_STR1 = 'H') AND (NB_FAIL_PURGE_REPURGE = 0 )THEN
							STEP_Regen := 'PURGE';
							STEP_REGEN_ID := 28 ;
							VAR_Affichage1 := INT_TO_STRING(STATE_Tps_restant);          
							VAR_Affichage2 := '';       
							VAR_Affichage3 := 'm';
							ID_ERREUR_REGEN := 1001;
							Regen_completed:=FALSE;
							VAR_Demande_Erreur:=FALSE;
						ELSIF (VAR_STR1 = 'H') AND (NB_FAIL_PURGE_REPURGE <> 0 )THEN
							STEP_Regen := 'REPURGE';
							STEP_REGEN_ID := 86 ;
							VAR_Affichage1 := CONCAT('#',UINT_TO_STRING(NB_FAIL_PURGE_REPURGE));          
							VAR_Affichage2 := INT_TO_STRING(STATE_Tps_restant);       
							VAR_Affichage3 := ' m';
							ID_ERREUR_REGEN := 1001;
							Regen_completed:=FALSE;
							VAR_Demande_Erreur:=FALSE;
						ELSIF (VAR_STR1 = 'I') OR (VAR_STR1 ='J')OR (VAR_STR1 = 'K') OR (VAR_STR1 ='T') THEN
							STEP_Regen := 'ROUGH TO BASE';
							STEP_REGEN_ID := 29 ;
							VAR_Affichage1 := REAL_TO_STRING(STATE_Pressure);          
							VAR_Affichage2 := 'u/';       
							VAR_Affichage3 := CONCAT(REAL_TO_STRING(PRM_RoughToPressure), 'μ');
							ID_ERREUR_REGEN := 1001;
							Regen_completed:=FALSE;
							VAR_Demande_Erreur:=FALSE;
						ELSIF (VAR_STR1 = 'L') THEN 
							STEP_Regen := 'ROR';
							STEP_REGEN_ID := 30 ;
							VAR_Affichage1 := CONCAT('#',INT_TO_STRING(STATE_ROR_nb));          
							VAR_Affichage2 := CONCAT(', ',INT_TO_STRING(LAST_ROR_Value));       
							VAR_Affichage3 := CONCAT('/',INT_TO_STRING(PRM_ROR));
							VAR_Affichage3 := CONCAT(VAR_Affichage3, ' μ/Min');
							ID_ERREUR_REGEN := 1001;
							Regen_completed:=FALSE;
							VAR_Demande_Erreur:=FALSE;
						ELSIF (VAR_STR1 = 'M') OR (VAR_STR1 ='N') THEN
							STEP_Regen := 'COOLDOWN';
							STEP_REGEN_ID := 31;
							VAR_Affichage1 := REAL_TO_STRING(STATE_Temperature[0]);          
							VAR_Affichage2 := '';       
							VAR_Affichage3 := '/17K';
							ID_ERREUR_REGEN := 1001;
							Regen_completed:=FALSE;
							VAR_Demande_Erreur:=FALSE;
						ELSIF (VAR_STR1 = 'W') THEN
							STEP_Regen := 'DELAY RESTART';
							STEP_REGEN_ID := 32;
							VAR_Affichage1 := REAL_TO_STRING(STATE_Tps_restant);          
							VAR_Affichage2 := '';       
							VAR_Affichage3 := 'm';
							ID_ERREUR_REGEN := 1001;
							Regen_completed:=FALSE;
							VAR_Demande_Erreur:=FALSE;
						ELSIF (VAR_STR1 = 'Z') THEN
							STEP_Regen := 'DELAY START';
							STEP_REGEN_ID := 33 ;
							VAR_Affichage1 := INT_TO_STRING(STATE_Tps_restant);          
							VAR_Affichage2 := '';       
							VAR_Affichage3 := 'm';
							ID_ERREUR_REGEN := 1001;
							Regen_completed:=FALSE;
							VAR_Demande_Erreur:=FALSE;
						ELSIF (VAR_STR1 = 'P') THEN
							STATE_Regen := FALSE;
							STEP_REGEN_ID := 34 ;
							IF iCounter_Evitement_1ere_requete_regen <> 0 THEN
								VAR_Mem_etape_Regen := FALSE;
							END_IF
							STEP_Regen := 'REGEN COMPLETED';
							Regen_completed:=TRUE;
							VAR_Demande_Erreur:=TRUE;
						ELSIF (VAR_STR1 = 'V') THEN
							STEP_Regen := 'REGEN ABORTED';
							STEP_REGEN_ID := 35;
							STATE_Regen := FALSE;
							VAR_Affichage1 := '';          
							VAR_Affichage2 := '';       
							VAR_Affichage3 := '';
							Regen_completed:=FALSE;
							VAR_Demande_Erreur:=TRUE;
						END_IF
						VAR_Affichage:= CONCAT(VAR_Affichage1, VAR_Affichage2);
						VAR_Affichage:=CONCAT(VAR_Affichage, VAR_Affichage3);
						
					1: (* demande température étage 2*)
						STATE_Temperature[1]	:=	STRING_TO_REAL(MID(VAR_TrameRetour,6,4));
					2:	(* demande pression*)
						STATE_Pressure	:=	STRING_TO_REAL(MID(VAR_TrameRetour,6,4));
					3:
							(* Demande erreur regen *)
						IF VAR_Demande_Erreur THEN
					 		VAR_STR1 :=	MID(VAR_TrameRetour,1,3);
							IF (VAR_STR1 = 'B') THEN 
								ID_ERREUR_REGEN := 58 ;
								REGEN_ERROR := 'WARMUP TIMEOUT';         (* garde pour debugger l'ID avec les textlist prend le dessus dans l'IHM*)
							ELSIF (VAR_STR1 = '@')AND (CO_Regen = FALSE) THEN
								ID_ERREUR_REGEN := 59;
								REGEN_ERROR := 'NO ERROR'; 
							ELSIF (VAR_STR1 = 'C') THEN
								ID_ERREUR_REGEN := 60;
								REGEN_ERROR := 'COOLDOWN TIMEOUT';
							ELSIF (VAR_STR1 = 'D') THEN
								ID_ERREUR_REGEN := 61;
								REGEN_ERROR := 'ERROR IN ROR';
							ELSIF (VAR_STR1 = 'E') THEN
								ID_ERREUR_REGEN := 62;
								REGEN_ERROR := 'ROR CYCLE LIMIT WAS REACHED';
							ELSIF (VAR_STR1 = 'F') THEN 
								ID_ERREUR_REGEN := 63;
								REGEN_ERROR := 'MANUAL ABORT';
							ELSIF (VAR_STR1 = 'G') THEN
								ID_ERREUR_REGEN := 64;
								REGEN_ERROR := 'ROUGH VALVE TIMEOUT';
							ELSIF (VAR_STR1 = 'H') THEN
								ID_ERREUR_REGEN := 65;
								REGEN_ERROR := 'system bug';
							ELSE
								ID_ERREUR_REGEN := 1001;
							END_IF
						END_IF	
					4:  (* tps restant pour les étapes avec une durée*)
						STATE_Tps_restant := STRING_TO_INT(MID(VAR_TrameRetour,3,4));
					5:  (*nb de test ROR effectué*)
						STATE_ROR_nb := STRING_TO_INT(MID(VAR_TrameRetour,2,4));
					6:
						LAST_ROR_Value := STRING_TO_INT(MID(VAR_TrameRetour,3,4));
					7:
						VAR_STR1	:=	MID(VAR_TrameRetour,1,3);
						STATE_Pompe	:=	(VAR_STR1 = '1');
					8: (* set rough valve*)
						VAR_STR1	:=	MID(VAR_TrameRetour,1,3);
						STATE_Rough_valve	:=	(VAR_STR1 = '1');
			
					9: (* set purge valve*)
						VAR_STR1	:=	MID(VAR_TrameRetour,1,3);
						STATE_Purge_valve	:=	(VAR_STR1 = '1');
					10: 
						NB_FAIL_PURGE_REPURGE	:=	STRING_TO_UINT(MID(VAR_TrameRetour,2,4));
					11: (* demande température étage 1*)
						STATE_Temperature[0]	:=	STRING_TO_REAL(MID(VAR_TrameRetour,6,4));
				END_CASE
				iCounter_Valeur_Num_Regen:= iCounter_Valeur_Num_Regen+1;
				IF iCounter_Valeur_Num_Regen>=12 THEN
					iCounter_Valeur_Num_Regen:=0;
				END_IF	
				iCounter_Evitement_1ere_requete_regen := iCounter_Evitement_1ere_requete_regen+1;
			15:
				VAR_Mem_CO_RoughValve_on	:=	FALSE;
				VAR_Mem_CO_RoughValve_off	:=	FALSE;
			16:
				VAR_Mem_CO_PurgeValve_on	:=	FALSE;
				VAR_Mem_CO_PurgeValve_off	:=	FALSE;
			
			17:
				CASE iCounter_Info_Pompe OF
					0:
						Pump_Serial_Number := MID(VAR_TrameRetour,8,3);
					1:
						Pump_Serial_Number_affiche := CONCAT(Pump_Serial_Number,MID(VAR_TrameRetour,4,3));
					2:
						Number_Of_Complete_Regen := STRING_TO_UINT(MID(VAR_TrameRetour,4,4));
					3:
						Time_Since_Last_Regen := STRING_TO_UINT(MID(VAR_TrameRetour,4,4));
					4:
						SoftwareRevisionLevel := MID(VAR_TrameRetour,7,3);
					5:
						ElaspedTime := STRING_TO_UINT(MID(VAR_TrameRetour,6,4));
				END_CASE
				iCounter_Info_Pompe:=iCounter_Info_Pompe+1;
				IF iCounter_Info_Pompe >=6 THEN
					iCounter_Info_Pompe:=0;
					VAR_Mem_CO_Info_Pompe := false;
				END_IF
				
			18: 
				VAR_Reception_Parametre := TRUE;
				VAR_Mem_CO_Envoie_Param_Relay := FALSE;
				
			19:
				TIMER_Delay_Relay.IN := PRM_Mode;
				TIMER_Delay_Relay.PT := UINT_TO_TIME(STRING_TO_UINT(VAR_Affichage_ValeurTIME_Relay)*1000);
				TIMER_Delay_Relay();
				IF TIMER_Delay_Relay.Q  THEN
					TAB_Affichage_Etat_Relay[PRM_Relay] := FALSE;
					PRM_Mode := FALSE;
				END_IF
				VAR_Reception_Parametre := TRUE;
				CASE iCounter_Param_Relay_lecture OF 
					0:
						VAR_Derniere_commande_Relay := MID(VAR_TrameRetour,1,3);
					1:
						VAR_Affichage_ValeurUL_Relay := lecture_valeur(VAR_TrameRetour);
					2: 
						VAR_Affichage_ValeurLL_Relay := lecture_valeur(VAR_TrameRetour);                 
					3:
						VAR_Affichage_ValeurTIME_Relay := lecture_valeur(VAR_TrameRetour);
				END_CASE
				iCounter_Param_Relay_lecture := iCounter_Param_Relay_lecture+1;
				IF iCounter_Param_Relay_lecture >= 4 THEN
					iCounter_Param_Relay_lecture := 0;
					VAR_Mem_CO_Lecture_Relay:=FALSE;
				END_IF
				IF VAR_Derniere_commande_Relay = '0' OR VAR_Derniere_commande_Relay = '1' THEN
					VAR_Affichage_Commande_Relay := 70;
					TIMER_Delay_Relay2.IN := Var_lancement_timer_ONOFF;
					TIMER_Delay_Relay2.PT := UINT_TO_TIME(STRING_TO_UINT(VAR_Affichage_ValeurTIME_Relay)*1000);
					TIMER_Delay_Relay2();
					IF TIMER_Delay_Relay2.Q  THEN
						TAB_Affichage_Etat_Relay[PRM_Relay] := FALSE;
						Var_lancement_timer_ONOFF := FALSE;
					END_IF
					TAB_Affichage_Mode_relay[PRM_Relay] := TRUE;
					VAR_Affichage_Valeur_Relay := CONCAT('LL=', VAR_Affichage_ValeurUL_Relay);
					VAR_Affichage_Valeur_Relay := CONCAT(VAR_Affichage_Valeur_Relay, '°K, UL=');
					VAR_Affichage_Valeur_Relay := CONCAT(VAR_Affichage_Valeur_Relay, VAR_Affichage_ValeurLL_Relay);
					VAR_Affichage_Valeur_Relay := CONCAT(VAR_Affichage_Valeur_Relay, '°K');
				ELSIF VAR_Derniere_commande_Relay = '2' OR VAR_Derniere_commande_Relay = '3' THEN
					VAR_Affichage_Commande_Relay := 71;
					TIMER_Delay_Relay2.IN := Var_lancement_timer_ONOFF;
					TIMER_Delay_Relay2.PT := UINT_TO_TIME(STRING_TO_UINT(VAR_Affichage_ValeurTIME_Relay)*1000);
					TIMER_Delay_Relay2();
					IF TIMER_Delay_Relay2.Q  THEN
						TAB_Affichage_Etat_Relay[PRM_Relay] := FALSE;
						Var_lancement_timer_ONOFF := FALSE;
					END_IF
					TAB_Affichage_Mode_relay[PRM_Relay] := TRUE;
					VAR_Affichage_Valeur_Relay := CONCAT('LL=', VAR_Affichage_ValeurUL_Relay);
					VAR_Affichage_Valeur_Relay := CONCAT(VAR_Affichage_Valeur_Relay, '°K, UL=');
					VAR_Affichage_Valeur_Relay := CONCAT(VAR_Affichage_Valeur_Relay, VAR_Affichage_ValeurLL_Relay);
					VAR_Affichage_Valeur_Relay := CONCAT(VAR_Affichage_Valeur_Relay, '°K');
				ELSIF VAR_Derniere_commande_Relay = '4' OR VAR_Derniere_commande_Relay = '5' THEN
					VAR_Affichage_Commande_Relay := 72;
					TIMER_Delay_Relay2.IN := Var_lancement_timer_ONOFF;
					TIMER_Delay_Relay2.PT := UINT_TO_TIME(STRING_TO_UINT(VAR_Affichage_ValeurTIME_Relay)*1000);
					TIMER_Delay_Relay2();
					IF TIMER_Delay_Relay2.Q  THEN
						TAB_Affichage_Etat_Relay[PRM_Relay] := FALSE;
						Var_lancement_timer_ONOFF := FALSE;
					END_IF
					TAB_Affichage_Mode_relay[PRM_Relay] := TRUE;
					VAR_Affichage_Valeur_Relay := CONCAT('LL=', VAR_Affichage_ValeurUL_Relay);
					VAR_Affichage_Valeur_Relay := CONCAT(VAR_Affichage_Valeur_Relay, 'u, UL=');
					VAR_Affichage_Valeur_Relay := CONCAT(VAR_Affichage_Valeur_Relay, VAR_Affichage_ValeurLL_Relay);
					VAR_Affichage_Valeur_Relay := CONCAT(VAR_Affichage_Valeur_Relay, 'u');
				ELSIF VAR_Derniere_commande_Relay = '6' OR VAR_Derniere_commande_Relay = '7' THEN
					VAR_Affichage_Commande_Relay := 73;
					TIMER_Delay_Relay2.IN := Var_lancement_timer_ONOFF;
					TIMER_Delay_Relay2.PT := UINT_TO_TIME(STRING_TO_UINT(VAR_Affichage_ValeurTIME_Relay)*1000);
					TIMER_Delay_Relay2();
					IF TIMER_Delay_Relay2.Q  THEN
						TAB_Affichage_Etat_Relay[PRM_Relay] := FALSE;
						Var_lancement_timer_ONOFF := FALSE;
					END_IF
					TAB_Affichage_Mode_relay[PRM_Relay] := TRUE;
					VAR_Affichage_Valeur_Relay := CONCAT('LL=', VAR_Affichage_ValeurUL_Relay);
					VAR_Affichage_Valeur_Relay := CONCAT(VAR_Affichage_Valeur_Relay, 'u, UL=');
					VAR_Affichage_Valeur_Relay := CONCAT(VAR_Affichage_Valeur_Relay, VAR_Affichage_ValeurLL_Relay);
					VAR_Affichage_Valeur_Relay := CONCAT(VAR_Affichage_Valeur_Relay, 'u');
				ELSIF VAR_Derniere_commande_Relay = '8' THEN
					VAR_Affichage_Commande_Relay := 74;
					VAR_Affichage_Valeur_Relay := CONCAT(VAR_Affichage_ValeurTIME_Relay, ' sec');
				ELSIF VAR_Derniere_commande_Relay = 'A' THEN
					VAR_Affichage_Commande_Relay := 75;
					TIMER_Delay_Relay2.IN := Var_lancement_timer_ONOFF;
					TIMER_Delay_Relay2.PT := UINT_TO_TIME(STRING_TO_UINT(VAR_Affichage_ValeurTIME_Relay)*1000);
					TIMER_Delay_Relay2();
					IF TIMER_Delay_Relay2.Q  THEN
						TAB_Affichage_Etat_Relay[PRM_Relay] := TRUE;
						Var_lancement_timer_ONOFF := FALSE;
					END_IF
					TAB_Affichage_Mode_relay[PRM_Relay] := FALSE;
					VAR_Affichage_Valeur_Relay := '';
				ELSIF VAR_Derniere_commande_Relay = 'B' THEN
					VAR_Affichage_Commande_Relay := 76;
					VAR_Affichage_Valeur_Relay := '';
					TIMER_Delay_Relay2.IN := Var_lancement_timer_ONOFF;
					TIMER_Delay_Relay2.PT := UINT_TO_TIME(STRING_TO_UINT(VAR_Affichage_ValeurTIME_Relay)*1000);
					TIMER_Delay_Relay2();
					IF TIMER_Delay_Relay2.Q  THEN
						TAB_Affichage_Etat_Relay[PRM_Relay] := FALSE;
						Var_lancement_timer_ONOFF := FALSE;
					END_IF
					TAB_Affichage_Mode_relay[PRM_Relay] := FALSE;
				ELSIF VAR_Derniere_commande_Relay = 'C' THEN
					VAR_Affichage_Commande_Relay := 77;
					TIMER_Delay_Relay2.IN := Var_lancement_timer_ONOFF;
					TIMER_Delay_Relay2.PT := UINT_TO_TIME(STRING_TO_UINT(VAR_Affichage_ValeurTIME_Relay)*1000);
					TIMER_Delay_Relay2();
					IF TIMER_Delay_Relay2.Q  THEN
						TAB_Affichage_Etat_Relay[PRM_Relay] := FALSE;
						Var_lancement_timer_ONOFF := FALSE;
					END_IF
					VAR_Affichage_Valeur_Relay := 'ON';
					TAB_Affichage_Mode_relay[PRM_Relay] := TRUE;
				ELSIF VAR_Derniere_commande_Relay = 'D' THEN
					VAR_Affichage_Commande_Relay := 78;
					TIMER_Delay_Relay2.IN := Var_lancement_timer_ONOFF;
					TIMER_Delay_Relay2.PT := UINT_TO_TIME(STRING_TO_UINT(VAR_Affichage_ValeurTIME_Relay)*1000);
					TIMER_Delay_Relay2();
					IF TIMER_Delay_Relay2.Q  THEN
						TAB_Affichage_Etat_Relay[PRM_Relay] := FALSE;
						Var_lancement_timer_ONOFF := FALSE;
					END_IF
					VAR_Affichage_Valeur_Relay := 'ON';
					TAB_Affichage_Mode_relay[PRM_Relay] := TRUE;
				ELSIF VAR_Derniere_commande_Relay = 'F' THEN
					VAR_Affichage_Commande_Relay := 79;
					VAR_Affichage_Valeur_Relay := 'ON';
					TIMER_Delay_Relay2.IN := Var_lancement_timer_ONOFF;
					TIMER_Delay_Relay2.PT := UINT_TO_TIME(STRING_TO_UINT(VAR_Affichage_ValeurTIME_Relay)*1000);
					TIMER_Delay_Relay2();
					IF TIMER_Delay_Relay2.Q  THEN
						TAB_Affichage_Etat_Relay[PRM_Relay] := FALSE;
						Var_lancement_timer_ONOFF := FALSE;
					END_IF
					TAB_Affichage_Mode_relay[PRM_Relay] := TRUE;
				END_IF
			20:
				iCounter_Param_ParDefaut_Relay_lecture:= iCounter_Param_ParDefaut_Relay_lecture+1;
				IF iCounter_Param_ParDefaut_Relay_lecture>=3 THEN
					iCounter_Param_ParDefaut_Relay_lecture:=0;
					VAR_Mem_CO_Param_usine_Relay:=false;
				END_IF
			21:
				VAR_Mem_CO_pumpTC_On	:=	FALSE;
				VAR_Mem_CO_pumpTC_Off	:=	FALSE;
		END_CASE

		(*trame suivante*)
		IF NOT CO_Forcage THEN
			IF VAR_Mem_CO_Off OR VAR_Mem_CO_On THEN
				VAR_Cadence := 11;
			ELSIF VAR_Mem_CO_RoughValve_On OR VAR_Mem_CO_RoughValve_Off THEN
				VAR_Cadence := 15;
			ELSIF VAR_Mem_CO_PurgeValve_On OR VAR_Mem_CO_PurgeValve_Off THEN
				VAR_Cadence := 16;
			ELSIF VAR_Mem_CO_pumpTC_On OR VAR_Mem_CO_pumpTC_Off THEN
				VAR_Cadence := 21;
			ELSIF VAR_Mem_CO_Ecriture THEN
				VAR_Cadence := 12;
			ELSIF VAR_Mem_CO_Lecture THEN
				VAR_Cadence := 13;
			ELSIF VAR_Mem_CO_Info_Pompe THEN
				VAR_Cadence := 17;
			ELSIF VAR_Mem_CO_Regen OR Var_Mem_CO_StopRegen THEN
				VAR_Cadence := 10;
			ELSIF VAR_Mem_Etape_Regen THEN
				VAR_Cadence := 14;
			ELSIF VAR_Mem_CO_Envoie_Param_Relay THEN
				VAR_Cadence := 18;
			ELSIF VAR_Mem_CO_Param_usine_Relay THEN
				VAR_Cadence := 20;
			ELSIF VAR_Mem_CO_Lecture_Relay THEN
				VAR_Cadence := 19;
			ELSE
				VAR_Cadence := VAR_Cadence + 1;
				IF VAR_Cadence >= 10 THEN
					VAR_Cadence	:=	1;
					STOP_LOAD:= TRUE;
				END_IF
			END_IF
		ELSE
			VAR_Cadence 	 := 	CONF_Forcage;
		END_IF
	ELSE
		IF CO_ModeManu THEN													(* gestion retour commande du mode manu*)
		IF PRM_TrameManu = 'A?' THEN
				(* Demande état On/off pompe *)
				VAR_STR1	:=	MID(VAR_TrameRetour,1,3);
				Reponse_ModeManu	:=	BOOL_TO_STRING((VAR_STR1 = '1'));
		ELSIF PRM_TrameManu = 'O' THEN
				(* Demande état regen pompe *)
				VAR_STR1	:=	MID(VAR_TrameRetour,1,3);
				IF (VAR_STR1 = 'B') OR (VAR_STR1 ='C')OR (VAR_STR1 = 'E') OR (VAR_STR1 ='Q') OR  (VAR_STR1 ='R') OR (VAR_STR1 ='^')  OR (VAR_STR1 =']') THEN 
					Reponse_ModeManu := 'WARM-UP'; 
				ELSIF (VAR_STR1 = 'D') OR (VAR_STR1 ='F')OR (VAR_STR1 = 'G') THEN
					Reponse_ModeManu := 'PURGE GAS FAILURE';
				ELSIF (VAR_STR1 = 'H') THEN
					Reponse_ModeManu := 'REPURGE';
				ELSIF (VAR_STR1 = 'I') OR (VAR_STR1 ='J')OR (VAR_STR1 = 'K') OR (VAR_STR1 ='T') THEN
					Reponse_ModeManu := 'ROUGH TO BASE';
				ELSIF (VAR_STR1 = 'L') THEN 
					Reponse_ModeManu := 'ROR';
				ELSIF (VAR_STR1 = 'M') OR (VAR_STR1 ='N') THEN
					Reponse_ModeManu := 'COULDOWN';
				ELSIF (VAR_STR1 = 'W') THEN
					Reponse_ModeManu := 'DELAY RESTART';
				ELSIF (VAR_STR1 = 'Z') THEN
					Reponse_ModeManu := 'DELAY START';
				ELSIF (VAR_STR1 = 'P') THEN
					Reponse_ModeManu := 'REGEN COMPLETED';
				ELSIF (VAR_STR1 = 'V') THEN
					Reponse_ModeManu := 'REGEN ABORTED';
				END_IF

		ELSIF PRM_TrameManu = 'J' THEN
				(* demande température étage 1*)
				Reponse_ModeManu	:=	REAL_TO_STRING(STRING_TO_REAL(MID(VAR_TrameRetour,6,4)));
		ELSIF PRM_TrameManu = 'K' THEN
				(* demande température étage 2*)
				Reponse_ModeManu	:=	REAL_TO_STRING(STRING_TO_REAL(MID(VAR_TrameRetour,6,4)));
		ELSIF PRM_TrameManu = 'L' THEN		
				(* demande pression*)
				Reponse_ModeManu	:=	REAL_TO_STRING(STRING_TO_REAL(MID(VAR_TrameRetour,6,4)));
		ELSIF PRM_TrameManu = 'e' THEN		
				(* Demande erreur regen *)
				VAR_STR1	:=	MID(VAR_TrameRetour,1,3);
				IF (VAR_STR1 = 'B') THEN 
					Reponse_ModeManu := 'WARMUP TIMEOUT';
				ELSIF (VAR_STR1 = '@') THEN
					Reponse_ModeManu := 'NO ERROR'; 
				ELSIF (VAR_STR1 = 'C') THEN
					Reponse_ModeManu := 'COOLDOWN TIMEOUT';
				ELSIF (VAR_STR1 = 'D') THEN
					Reponse_ModeManu := 'ERROR IN ROR';
				ELSIF (VAR_STR1 = 'E') THEN
					Reponse_ModeManu := 'ROR CYCLE LIMIT WAS REACHED';
				ELSIF (VAR_STR1 = 'F') THEN 
					Reponse_ModeManu := 'MANUAL ABORT';
				ELSIF (VAR_STR1 = 'G') THEN
					REGEN_ERROR := 'ROUGH VALVE TIMEOUT';
				ELSIF (VAR_STR1 = 'H') THEN
					Reponse_ModeManu := 'system bug';
				END_IF
				
		ELSIF PRM_TrameManu ='P1?' OR PRM_TrameManu ='P0?'OR PRM_TrameManu ='P2?'OR PRM_TrameManu ='P3?'OR PRM_TrameManu ='P4?'OR PRM_TrameManu ='P5?' OR PRM_TrameManu = 'P6?' OR PRM_TrameManu = 'PA?'  OR PRM_TrameManu = 'PG?' OR PRM_TrameManu = 'i?' OR PRM_TrameManu = 'j?'THEN					
				(* Demande lecture parametre regen pompe en mode manuel *)
				IF MID(PRM_TrameManu,1,2)='A' THEN
					Reponse_ModeManu := BOOL_TO_STRING(STRING_TO_BOOL(MID(VAR_TrameRetour,1,3)));
				ELSIF MID(PRM_TrameManu,1,2)= 'G' THEN
					Reponse_ModeManu := USINT_TO_STRING(STRING_TO_USINT(MID(VAR_TrameRetour,4,4)));
				ELSIF MID(PRM_TrameManu,1,1)= 'i' THEN
					Reponse_ModeManu := USINT_TO_STRING(STRING_TO_USINT(MID(VAR_TrameRetour,1,3)));
				ELSIF MID(PRM_TrameManu,1,1)= 'j' THEN
					Reponse_ModeManu := USINT_TO_STRING(STRING_TO_USINT(MID(VAR_TrameRetour,4,4)));
				ELSE
					iCounter_ModeManu_lectureRegen := STRING_TO_INT(MID(PRM_TrameManu,1,3));
				CASE iCounter_ModeManu_lectureRegen OF 
					0: 
						Reponse_ModeManu :=	UINT_TO_STRING(STRING_TO_UINT(MID(VAR_TrameRetour,5,4)));                   (*ajouter la fonction lecture valeur*)
					1:
						Reponse_ModeManu := UINT_TO_STRING(STRING_TO_UINT(MID(VAR_TrameRetour,4,4)));
					2:
						Reponse_ModeManu  := USINT_TO_STRING(STRING_TO_USINT(MID(VAR_TrameRetour,2,4)));
					3:
						Reponse_ModeManu  :=USINT_TO_STRING(STRING_TO_USINT(MID(VAR_TrameRetour,3,4)));
					4:
						Reponse_ModeManu := USINT_TO_STRING(STRING_TO_USINT(MID(VAR_TrameRetour,3,4)));
					5:
						Reponse_ModeManu := USINT_TO_STRING(STRING_TO_USINT(MID(VAR_TrameRetour,2,4))); 
					6:
						Reponse_ModeManu := UINT_TO_STRING(STRING_TO_UINT(MID(VAR_TrameRetour,6,4)));
				END_CASE
				END_IF
			ELSIF PRM_TrameManu = 'D?'  THEN	
				(* read rough valve*)
				VAR_STR1	:=	MID(VAR_TrameRetour,1,3);
				Reponse_ModeManu	:=	BOOL_TO_STRING(VAR_STR1 = '1');
			ELSIF PRM_TrameManu = 'E?'  THEN	
				(* read purge valve*)
				VAR_STR1	:=	MID(VAR_TrameRetour,1,3);
				Reponse_ModeManu	:=	BOOL_TO_STRING(VAR_STR1 = '1');
			ELSIF PRM_TrameManu = 'N1' OR PRM_TrameManu = 'N0' THEN		
				(* Demande de regen ou arrêt regen d'une pompe *)
				VAR_Mem_CO_StopRegen	:=	FALSE;
				VAR_Mem_CO_Regen	:=	FALSE;
				Reponse_ModeManu := 'Ok';
			ELSIF PRM_TrameManu = 'A1' OR PRM_TrameManu = 'A0' THEN		
				(* Demande de marche ou d'arrêt d'une pompe *)
				VAR_Mem_CO_Off	:=	FALSE;
				VAR_Mem_CO_On	:=	FALSE;
				Reponse_ModeManu := 'Ok';
			ELSIF MID(PRM_TrameManu,1,1) = 'P' OR MID(PRM_TrameManu,1,1) = 'i' OR MID(PRM_TrameManu,1,1) = 'j'   THEN	
				VAR_Reception_Parametre := TRUE;
				IF iCounter_Regen_ecriture = 0 THEN 
					VAR_Mem_CO_Ecriture := FALSE;
				END_IF
				Reponse_ModeManu := 'Ok';
			ELSIF PRM_TrameManu = 'D1' OR PRM_TrameManu ='D0' THEN	
				VAR_Mem_CO_RoughValve_on	:=	FALSE;
				VAR_Mem_CO_RoughValve_off	:=	FALSE;
				Reponse_ModeManu := 'Ok';
			ELSIF PRM_TrameManu = 'E1' OR PRM_TrameManu ='E0' THEN	
				VAR_Mem_CO_PurgeValve_on	:=	FALSE;
				VAR_Mem_CO_PurgeValve_off	:=	FALSE;
				Reponse_ModeManu := 'Ok';
			
			ELSIF PRM_TrameManu = 'Z?'  THEN
				Reponse_ModeManu := UINT_TO_STRING(STRING_TO_UINT(MID(VAR_TrameRetour,4,4)));
			ELSIF PRM_TrameManu = 'VA?'  THEN
				Reponse_ModeManu := MID(VAR_TrameRetour,8,3);
			ELSIF PRM_TrameManu = 'VQ?'  THEN
				Reponse_ModeManu := MID(VAR_TrameRetour,4,3);
			ELSIF PRM_TrameManu = 'Y?'  THEN
				Reponse_ModeManu := UINT_TO_STRING(STRING_TO_UINT(MID(VAR_TrameRetour,6,4)));
			ELSIF PRM_TrameManu = 'a'  THEN
				Reponse_ModeManu := UINT_TO_STRING(STRING_TO_UINT(MID(VAR_TrameRetour,4,4)));
			ELSIF PRM_TrameManu = '@'  THEN
				Reponse_ModeManu := MID(VAR_TrameRetour,7,3);
			END_IF
		END_IF
	END_IF

	VAR_ReceptionOk := TRUE;

	(*Effacement buffer réception*)
	VAR_ClearBuffer(Buffer := IN_Buffer);
END_IF

(* GESTION COMMUNICATION *)
VAR_COMportControl(
	Mode:= SERIALLINEMODE_PC_COM_PORT,
	pComIn:= ADR(IN_COM),
	pComOut:= ADR(OUT_COM),
	SizeComIn:=SIZEOF(IN_COM),
	TxBuffer:= OUT_Buffer,
	RxBuffer:= IN_Buffer,
	Error=> VAR_COMportControlError,
	ErrorID=> VAR_COMportControlErrorID );

(*GESTION DEFAUTS*)
Def_port_com.DELAY :=T#0s;
Def_port_com.CONDITION := VAR_COMportControlError;
Def_port_com();

(*Etat*)
STATE_Ready		:=	NOT OFF;
STATE_NOK		:=	Def_port_com.DEF;

END_FUNCTION_BLOCK

// ---- POUs/Fonction/FONCTIONS UTILITAIRES/CHECKSUM.TcPOU
FUNCTION CHECKSUM : STRING

VAR_INPUT
	PRM_CHR:			STRING;
	PRM_AvecDollars:	BOOL;
END_VAR

VAR
	VAR_STR:		STRING(1);
	VAR_NB:			BYTE;
	VAR_Somme1:		BYTE;
	VAR_Somme2:		BYTE;
	VAR_Somme3:		BYTE;
END_VAR

VAR_STR	:=	'X';
IF PRM_AvecDollars THEN
	VAR_NB		:=	2;
ELSE
	VAR_NB		:=	1;
END_IF
VAR_Somme1	:=	0;
WHILE VAR_STR <> '' DO
	VAR_STR	:=	MID(STR:=PRM_CHR, LEN:=1, POS:=VAR_NB);
	IF VAR_STR <> '' THEN
		VAR_Somme1	:=	VAR_Somme1 + ASC(VAR_STR);
	END_IF
	VAR_NB		:=	VAR_NB + 1;
END_WHILE

(*Somme2	:=	ROR(Somme1,6);*)
VAR_NB		:=	0;
VAR_NB.0	:=	VAR_Somme1.6;
VAR_NB.1	:=	VAR_Somme1.7;
(*Somme2	:=	2;*)
VAR_Somme3	:=	VAR_Somme1 XOR VAR_NB;
VAR_Somme1	:=	63;
VAR_Somme3	:=	VAR_Somme3 AND VAR_Somme1;
VAR_Somme2	:=	VAR_Somme3 + 48;

CHECKSUM	:=	CHR(VAR_Somme2);
RETURN;

END_FUNCTION

// ---- POUs/Composant/POMPES/CRYO CTI/Lecture_valeur.TcPOU
FUNCTION Lecture_valeur :STRING
VAR_INPUT
	VAR_Trame_entiere:	STRING;
END_VAR
VAR_OUTPUT
	VAR_Trame_valeur:   STRING:= '';
END_VAR
VAR
	VAR_STR:   STRING(1):='0';
	VAR_Compteur: INT:= 4;
	VAR_Trame_CHECKSUM: STRING:='';
	VAR_CHECKSUM: STRING;
END_VAR


VAR_Trame_CHECKSUM := MID(VAR_Trame_entiere, LEN:=3, POS:=1);
WHILE (VAR_STR <>'') DO
	VAR_STR	:=	MID(VAR_Trame_entiere, LEN:=1, POS:=VAR_Compteur);
	VAR_CHECKSUM := CHECKSUM(VAR_Trame_CHECKSUM, TRUE);
	IF VAR_STR <> VAR_CHECKSUM THEN
		VAR_Trame_valeur := CONCAT(VAR_Trame_valeur,VAR_STR);
		VAR_Trame_CHECKSUM:= CONCAT(VAR_Trame_CHECKSUM,VAR_STR);
		VAR_Compteur := VAR_Compteur+1;
	END_IF
	IF VAR_STR = VAR_CHECKSUM THEN
		VAR_Compteur:=4;
		VAR_STR:='';
	END_IF

END_WHILE
VAR_STR:= MID(VAR_Trame_valeur,LEN:=1,POS:=1);
WHILE (VAR_STR = '0') DO
	VAR_STR:= MID(VAR_Trame_valeur,LEN:=1,POS:=1);
	IF (VAR_STR = '0') THEN
		VAR_Trame_valeur := DELETE(VAR_Trame_valeur,LEN:=1,POS:=1);
	END_IF
END_WHILE
IF VAR_Trame_valeur ='' THEN
	VAR_Trame_valeur :='0';
END_IF
Lecture_valeur := VAR_Trame_valeur;
RETURN;

END_FUNCTION

// ---- POUs/Programme/BLOCK_PRG_SERVITUDES.TcPOU
FUNCTION_BLOCK BLOCK_PRG_SERVITUDES

(*****************************************************************)
(* 		Programme servitudes
		PRG_SERVITUDES_8LIGNES_SIMPLES
		Gestion jusqu'à 8 lignes d'eau simple			      
 		Gestion de la commutation eau chaude / eau froide 
		Version 0 - HG - 03/2011                                     
		FAMILLE : CT200								     *)
(*****************************************************************)
VAR_INPUT
	//IN_GF1OK		AT%I*:		BOOL;		(*Entrée défaut circulateur eau*)
	//IN_GF1NivCh		AT%I*:		BOOL;		(*Entrée niveau haut eau chaude*)
	//IN_C1T			AT%I*:		BOOL;		(*Entree de détection de fuite enceinte*)

	IN_DE1T			AT%I*:		BOOL;
	IN_DE2T			AT%I*:		BOOL;
	IN_DE3T			AT%I*:		BOOL;
	IN_DE5T			AT%I*:		BOOL;
	IN_DE4T			AT%I*:		BOOL;
	IN_DE6T			AT%I*:		BOOL;
	IN_DE7T			AT%I*:		BOOL;
	IN_DE8T			AT%I*:		BOOL;

	
	LIGNE_REF:				ARRAY[1..8] OF BLOCK_LIGNE_REF;	

	EAU:						BLOCK_WREFCH1;

	DEF_Groupe:					PRCDEF;	(*Défaut du groupe chaud/froid*)
	DEF_Fuite:					PRCDEF;	(*Défaut de détection d'une fuite dans l'enceinte*)

END_VAR

VAR_INPUT PERSISTENT
	CONF_CO_ON:			ARRAY[0..8] OF USINT;	(*Indique quelle condition déclenche la mise en marche de la circulation d'eau froide
															0 = condition de mise en marche = condition de refroidissement impératif
															1 = condition de vide dans l'enceinte
															2 = reserve 
															3 = mise en marche de la machine
															*)
	PRM_Pr_REF_ENC:			REAL;					(* I_STANDARD --- Pression de mise en marche du refroidissement pour les élément lié à l'enceinte *)
	PRM_Forcage_Chaud:		BOOL;					(*Forcage circulation eau chaude*)

	PRM_tps_att_chaud:		TIME;					(*temps d'attente avant obtention état chaud*)

	CONF_eau_chaude:		BOOL;					(*indique la présence d'un commutateur eau chaude / eau froide*)

	(*Entité*)
	IsAssembly:		BOOL;			(*entité : assembly*)
	IdXML:			STRING;			(*nom entité : identifiant pour recherche dans dico*)
	TagXML:			UINT;			(*nom entité : identifiant pour recherche dans dico*)
	IdParent:			STRING;			(*MNEMO de l'appelant*)
	MNEMO:			STRING;			(*MNEMO de l'entité*)
END_VAR

VAR_OUTPUT
	OUT_VE1			AT%Q*:		BOOL;
	OUT_VE2			AT%Q*:		BOOL;
	OUT_VE3			AT%Q*:		BOOL;
	OUT_VE4			AT%Q*:		BOOL;
	OUT_VE5			AT%Q*:		BOOL;
	OUT_VE6			AT%Q*:		BOOL;
	OUT_VE7			AT%Q*:		BOOL;
	OUT_VE8			AT%Q*:		BOOL;

	(*vannes circulation eau chaude eau froide*)
	OUT_VEC11			AT%Q*:		BOOL;
	OUT_VEF11			AT%Q*:		BOOL;
	OUT_VEC12			AT%Q*:		BOOL;
	OUT_VEF12			AT%Q*:		BOOL;

	OUT_GF1			AT%Q*:		BOOL;	(*Mise en marche compresseur eau chaude*)
	OUT_MGF1		AT%Q*:		BOOL;	(*Mise en puissance compresseur pour eco-mode*)

	WATER:		ARRAY[0..8] OF BOOL;			(* I_STANDARD --- information de débit d'eau pour chaque ligne*)
	STATE_AR:	ARRAY[0..8] OF BOOL;			(* I_STANDARD ---information de débit d'eau stoppé pour chaque ligne*)
END_VAR

VAR
	I:						USINT;
	TIMER_chaud:			TON;		(*timer obtention état chaud*)
	FM_state_chaud:			R_TRIG;		(*front montant etat chaud*)
	var_mem_prep_ventil:	BOOL;		(*mémorisation de la demande de préparation de ventilation*)
	var_state_froid:		BOOL;		(*état eau froide en cours, utile si pas eau chaude (ds ce cas state froid n'est pas maj par EAU)*)
	STATE_Manu:				BOOL;		(*Recopie de l'information ENCEINTE.STATE_Manu*)
	FM_Etape_Pompage_OK: 	R_TRIG;
	FM_RQ_Start_Prod:		R_TRIG;
	FM_RQ_Stop_Prod:		R_TRIG;
END_VAR

(*Recopie*)
STATE_Manu			:=	MACHINE.STATE_Manu;

(*Reset des ordres de forçage eau chaude*)
FM_Etape_Pompage_OK(clk:= PRG_POMPAGE.O_STEP_PUMPING_OK );
FM_RQ_Start_Prod(clk:= MACHINE.RQ_Start_Prod);
FM_RQ_Stop_Prod(clk:= MACHINE.RQ_Stop_Prod);

IF FM_RQ_Start_Prod.Q OR FM_RQ_Stop_Prod.Q OR MACHINE.STATE_Off OR MACHINE.STATE_Manu
OR FM_Etape_Pompage_OK.Q OR EAU.OP_CHAUD.DEF_AUTO_ON.DEF OR EAU.OP_CHAUD.DEF_ON_REJECTED.DEF  THEN
	PRM_Forcage_Chaud 	:= 	FALSE;
END_IF

(*General*)
IdXML								:=		'6';
TagXML								:=		0;

(*Parametre statique*)
CONF_eau_chaude						:=		FALSE;
PRM_Pr_REF_ENC						:=		0.1;

LIGNE_REF[1].DEF_Ref.DELAY			:=		T#5S;
LIGNE_REF[2].DEF_Ref.DELAY			:=		T#5S;
LIGNE_REF[3].DEF_Ref.DELAY			:=		T#5S;
LIGNE_REF[4].DEF_Ref.DELAY			:=		T#5S;
LIGNE_REF[5].DEF_Ref.DELAY			:=		T#5S;
LIGNE_REF[6].DEF_Ref.DELAY			:=		T#5S;
LIGNE_REF[7].DEF_Ref.DELAY			:=		T#5S;
LIGNE_REF[8].DEF_Ref.DELAY			:=		T#5S;

LIGNE_REF[1].CONF_TIM_OFF			:=		T#60S;
LIGNE_REF[2].CONF_TIM_OFF			:=		T#60S;
LIGNE_REF[3].CONF_TIM_OFF			:=		T#60S;
LIGNE_REF[4].CONF_TIM_OFF			:=		T#60S;
LIGNE_REF[5].CONF_TIM_OFF			:=		T#60S;
LIGNE_REF[6].CONF_TIM_OFF			:=		T#60S;
LIGNE_REF[7].CONF_TIM_OFF			:=		T#60S;
LIGNE_REF[8].CONF_TIM_OFF			:=		T#60S;


LIGNE_REF[1].CONF_NO_DexT			:=		FALSE;
LIGNE_REF[2].CONF_NO_DexT			:=		FALSE;
LIGNE_REF[3].CONF_NO_DexT			:=		FALSE;
LIGNE_REF[4].CONF_NO_DexT			:=		FALSE;
LIGNE_REF[5].CONF_NO_DexT			:=		TRUE;
LIGNE_REF[6].CONF_NO_DexT			:=		TRUE;
LIGNE_REF[7].CONF_NO_DexT			:=		TRUE;
LIGNE_REF[8].CONF_NO_DexT			:=		TRUE;

LIGNE_REF[1].CONF_No_Def_Dex		:= 		TRUE;
LIGNE_REF[2].CONF_No_Def_Dex		:=		TRUE;
LIGNE_REF[3].CONF_No_Def_Dex		:= 		TRUE;
LIGNE_REF[4].CONF_No_Def_Dex		:=		TRUE;
LIGNE_REF[5].CONF_No_Def_Dex		:=		TRUE;
LIGNE_REF[6].CONF_No_Def_Dex		:=		TRUE;
LIGNE_REF[7].CONF_No_Def_Dex		:=		TRUE;
LIGNE_REF[8].CONF_No_Def_Dex		:=		TRUE;

LIGNE_REF[1].MNEMO_Dex				:=		'DE1T';
LIGNE_REF[2].MNEMO_Dex				:=		'DE2T';
LIGNE_REF[3].MNEMO_Dex				:=		'DE3T';
LIGNE_REF[4].MNEMO_Dex				:=		'DE4T';
LIGNE_REF[5].MNEMO_Dex				:=		'DE5T';
LIGNE_REF[6].MNEMO_Dex				:=		'DE6T';
LIGNE_REF[7].MNEMO_Dex				:=		'DE7T';
LIGNE_REF[8].MNEMO_Dex				:=		'DE8T';

LIGNE_REF[1].VEx.MNEMO				:=		'VE1';
LIGNE_REF[2].VEx.MNEMO				:=		'VE2';
LIGNE_REF[3].VEx.MNEMO				:=		'VE3';
LIGNE_REF[4].VEx.MNEMO				:=		'VE4';
LIGNE_REF[5].VEx.MNEMO				:=		'VE5';
LIGNE_REF[6].VEx.MNEMO				:=		'VE6';
LIGNE_REF[7].VEx.MNEMO				:=		'VE7';
LIGNE_REF[8].VEx.MNEMO				:=		'VE8';

LIGNE_REF[1].MNEMO					:=		'Quartz';
LIGNE_REF[2].MNEMO					:=		'EJ-Gauche';
LIGNE_REF[3].MNEMO					:=		'EJ-Droite';
LIGNE_REF[4].MNEMO					:=		'Canon e-';
LIGNE_REF[5].MNEMO					:=		'ACG600';
LIGNE_REF[6].MNEMO					:=		'Ligne 6';
LIGNE_REF[7].MNEMO					:=		'Ligne 7';
LIGNE_REF[8].MNEMO					:=		'Ligne 8';

LIGNE_REF[1].TagXML					:=		3;
LIGNE_REF[2].TagXML					:=		4;
LIGNE_REF[3].TagXML					:=		5;
LIGNE_REF[4].TagXML					:=		6;
LIGNE_REF[5].TagXML					:=		7;
LIGNE_REF[6].TagXML					:=		8;
LIGNE_REF[7].TagXML					:=		9;
LIGNE_REF[8].TagXML					:=		10;

FOR I:= 1 TO 7 DO
	LIGNE_REF[I].IdXML					:=	'6';
END_FOR;

DEF_Groupe.IdXML						:=	'8';
DEF_Groupe.TagXML						:=	3;

DEF_Fuite.IdXML							:=	'14';
DEF_Fuite.TagXML						:=	18;

CONF_CO_ON[1]							:=	3;
CONF_CO_ON[2]							:=	0;
CONF_CO_ON[3]							:=	0;
CONF_CO_ON[4]							:=	0;
CONF_CO_ON[5]							:=	0;
CONF_CO_ON[6]							:=	0;
CONF_CO_ON[7]							:=	0;
CONF_CO_ON[8]							:=	0;

EAU.VEC_IN.MNEMO						:=	'VEH1';
EAU.VEC_OUT.MNEMO						:=	'VEH2';
EAU.VEF_IN.MNEMO						:=	'VEC1';
EAU.VEF_OUT.MNEMO						:=	'VEC2';

(*************************************************************************************)
(*                          Gestion eau chaude / eau froide                          *)
(*************************************************************************************)
 (*mise en eau chaude en demande de préparation à la ventilation ou lorsque l'enceinte est à atmosphère*)
IF 	(PRG_POMPAGE.RQ_PREP_VENTIL OR PRG_POMPAGE.M11.STATE_Seuil[1] OR PRM_Forcage_Chaud) AND NOT STATE_Manu AND CONF_eau_chaude THEN
	EAU.OP_CHAUD.ON_PLC		:=	TRUE;
	EAU.OP_FROID.ON_PLC		:=	FALSE;
(*mise en eau froide à partir du seuil de pression défini par PRM_Pr_ref_enc (passé dans M11) *)
ELSIF PRG_POMPAGE.O_REF_ENC AND NOT PRM_Forcage_Chaud  AND NOT STATE_Manu AND CONF_eau_chaude THEN
	EAU.OP_CHAUD.ON_PLC	:= 	FALSE;
	EAU.OP_FROID.ON_PLC	:= 	TRUE;
END_IF
(*EAU(
	RESET:= 			MACHINE.STATE_off,
	MANUAL:= 			STATE_Manu,
	CTRL_PLC:=			TRUE ,						(*toujours piloté par l'automate*)
	CONF_Tim_Step:= 	T#5s,
	IN_NIV:=			IN_GF1NivCh,
	);
*)
(*mémorisation de la demande de préparation de ventilation*)
IF PRG_POMPAGE.RQ_PREP_VENTIL OR PRM_Forcage_Chaud THEN  (*mémo à la réception de la demande*)
	var_mem_prep_ventil := TRUE;
ELSIF NOT PRG_POMPAGE.POMPAGE.OP_Ventilation.EC AND NOT PRM_Forcage_Chaud THEN (*annulation lorsque plus ventilation en cours ou reset*)
	var_mem_prep_ventil := FALSE;
END_IF

(*renseignement de l'état eau froide*)
IF CONF_eau_chaude THEN
	var_state_froid := EAU.STATE_Froid;
ELSE
	var_state_froid := TRUE;
END_IF

(* 	Paramètre contextuel	*)
LIGNE_REF[1].I_Cond_need_Ref		:=		PRG_POMPAGE.RQ_REF[1];
LIGNE_REF[2].I_Cond_need_Ref		:=		PRG_EVAP.EVAPS2.RQ_Ref_source;
LIGNE_REF[3].I_Cond_need_Ref		:=		PRG_EVAP.EVAPS3.RQ_Ref_source;
LIGNE_REF[4].I_Cond_need_Ref		:=		PRG_EVAP.EVAPS1.RQ_Ref_source;
LIGNE_REF[5].I_Cond_need_Ref		:=		PRG_POMPAGE.RQ_REF[5];
LIGNE_REF[6].I_Cond_need_Ref		:=		PRG_POMPAGE.RQ_REF[6];
LIGNE_REF[7].I_Cond_need_Ref		:=		PRG_POMPAGE.RQ_REF[7];
LIGNE_REF[8].I_Cond_need_Ref		:=		PRG_POMPAGE.RQ_REF[8];

FOR I:=1 TO 8 DO
	//LIGNE_REF[I].I_Cond_need_Ref	:=		PRG_POMPAGE.RQ_REF[I];
	LIGNE_REF[I].CO_On				:=		((CONF_CO_ON[I] = 0) AND LIGNE_REF[I].I_Cond_need_Ref) OR
											((CONF_CO_ON[I] = 1) AND (PRG_POMPAGE.O_REF_ENC
											OR (var_mem_prep_ventil AND CONF_eau_chaude))) OR (CONF_CO_ON[I] = 3 AND OUT_MGF1);	
END_FOR;


(*************************************************************************************)
(*                                       Groupe froid					                              *)
(*************************************************************************************)
(*DEF_Groupe(
	CONDITION:= 	NOT IN_GF1OK AND NOT MACHINE.STATE_Off AND FALSE, //SPEC 14035
	DELAY:= 		T#5s
);
*)
(*************************************************************************************)
(*                                       Fuite enceinte					                              *)
(*************************************************************************************)
(*DEF_Fuite.CONDITION	:=	NOT IN_C1T AND NOT MACHINE.STATE_Off AND FALSE; //SPEC 14035
DEF_Fuite.DELAY		:=	T#2S;
DEF_Fuite();

*)
(*************************************************************************************)
(*                                       Ligne 1						                              *)
(*************************************************************************************)
LIGNE_REF[1].VEx.EN_On_EXT := NOT DEF_Fuite.DEF; (*Arrêt automatique si fuite détectée d'eau dans l'enceinte*)
LIGNE_REF[1]
	(
	RESET:= 				MACHINE.STATE_Off,
	MANUAL:=				STATE_Manu,
	I_inhibe_surv_ref:=		NOT var_state_froid ,
	I_Cond_Ref_Ok:=			var_state_froid AND NOT DEF_Groupe.DEF,
	IN_DExT:=				IN_DE1T,
	);

(*************************************************************************************)
(*                                       		Ligne 2							           *)
(*************************************************************************************)
LIGNE_REF[2].VEx.EN_On_EXT := NOT DEF_Fuite.DEF; (*Arrêt automatique si fuite détectée d'eau dans l'enceinte*)
LIGNE_REF[2]
	(
	RESET:= 				MACHINE.STATE_Off,
	MANUAL:=				STATE_Manu ,
	I_inhibe_surv_ref:=		NOT var_state_froid,
	I_Cond_Ref_Ok:=			var_state_froid AND NOT DEF_Groupe.DEF,
	IN_DExT:=				IN_DE2T,
	);

(*************************************************************************************)
(*                                     		 Ligne 3								 *)
(*************************************************************************************)
LIGNE_REF[3].VEx.EN_On_EXT := NOT DEF_Fuite.DEF; (*Arrêt automatique si fuite détectée d'eau dans l'enceinte*)
LIGNE_REF[3]
	(
	RESET:= 				MACHINE.STATE_Off,
	MANUAL:=				STATE_Manu ,
	I_inhibe_surv_ref:=		NOT var_state_froid ,
	I_Cond_Ref_Ok:=			var_state_froid AND NOT DEF_Groupe.DEF,
	IN_DExT:=				IN_DE3T,
	);

(*************************************************************************************)
(*                                     		 Ligne 4								 *)
(*************************************************************************************)
LIGNE_REF[4].VEx.EN_On_EXT := NOT DEF_Fuite.DEF; (*Arrêt automatique si fuite détectée d'eau dans l'enceinte*)
LIGNE_REF[4]
	(
	RESET:= 				MACHINE.STATE_Off,
	MANUAL:=				STATE_Manu ,
	I_inhibe_surv_ref:=		NOT var_state_froid ,
	I_Cond_Ref_Ok:=			var_state_froid AND NOT DEF_Groupe.DEF,
	IN_DExT:=				IN_DE4T,
	);

(*************************************************************************************)
(*                                     		 Ligne 5								 *)
(*************************************************************************************)
LIGNE_REF[5].VEx.EN_On_EXT := NOT DEF_Fuite.DEF; (*Arrêt automatique si fuite détectée d'eau dans l'enceinte*)
LIGNE_REF[5]
	(
	RESET:= 				MACHINE.STATE_Off,
	MANUAL:=				STATE_Manu ,
	I_inhibe_surv_ref:=		NOT var_state_froid ,
	I_Cond_Ref_Ok:=			var_state_froid AND NOT DEF_Groupe.DEF,
	//IN_DExT:=				IN_DE5T,
	);
	
(*************************************************************************************)
(*                                     		 Ligne 6								 *)
(*************************************************************************************)
LIGNE_REF[6].VEx.EN_On_EXT := NOT DEF_Fuite.DEF; (*Arrêt automatique si fuite détectée d'eau dans l'enceinte*)
LIGNE_REF[6]
	(
	RESET:= 				MACHINE.STATE_Off,
	MANUAL:=				STATE_Manu ,
	I_inhibe_surv_ref:=		NOT var_state_froid ,
	I_Cond_Ref_Ok:=			var_state_froid AND NOT DEF_Groupe.DEF,
	//IN_DExT:=				IN_DE6T,
	);
	
(*************************************************************************************)
(*                                     		 Ligne 7								 *)
(*************************************************************************************)
LIGNE_REF[7].VEx.EN_On_EXT := NOT DEF_Fuite.DEF; (*Arrêt automatique si fuite détectée d'eau dans l'enceinte*)
LIGNE_REF[7]
	(
	RESET:= 				MACHINE.STATE_Off,
	MANUAL:=				STATE_Manu ,
	I_inhibe_surv_ref:=		NOT var_state_froid ,
	I_Cond_Ref_Ok:=			var_state_froid AND NOT DEF_Groupe.DEF,
	//IN_DExT:=				IN_DE7T,
	);
	
(*************************************************************************************)
(*                                     		 Ligne 8								 *)
(*************************************************************************************)
LIGNE_REF[8].VEx.EN_On_EXT := NOT DEF_Fuite.DEF; (*Arrêt automatique si fuite détectée d'eau dans l'enceinte*)
LIGNE_REF[8]
	(
	RESET:= 				MACHINE.STATE_Off,
	MANUAL:=				STATE_Manu ,
	I_inhibe_surv_ref:=		NOT var_state_froid ,
	I_Cond_Ref_Ok:=			var_state_froid AND NOT DEF_Groupe.DEF,
	//IN_DExT:=				IN_DE8T,
	);

(*	Affectation des sorties	*)
OUT_VE1		:=	LIGNE_REF[1].VEx.OUT_On;
OUT_VE2		:=	LIGNE_REF[2].VEx.OUT_On;
OUT_VE3		:=	LIGNE_REF[3].VEx.OUT_On;
OUT_VE4		:=	LIGNE_REF[4].VEx.OUT_On;
OUT_VE5		:=	LIGNE_REF[5].VEx.OUT_On;
OUT_VE6		:=	LIGNE_REF[6].VEx.OUT_On;
OUT_VE7		:=	LIGNE_REF[7].VEx.OUT_On;
OUT_VE8		:=	LIGNE_REF[8].VEx.OUT_On;

OUT_VEC11		:=	EAU.VEC_IN.OUT_On;
OUT_VEC12		:=	EAU.VEC_OUT.OUT_On;
OUT_VEF11		:=	EAU.VEF_IN.OUT_On;
OUT_VEF12		:=	EAU.VEF_OUT.OUT_On;

OUT_GF1			:=	(OUT_VEC11 AND OUT_VEC12) OR (OUT_VEC11 AND OUT_VEF12);																										(*Mise en marche du compresseur eau chaude*)
OUT_MGF1		:=	NOT PRG_EVAP.ECO_MODE OR NOT PRG_POMPAGE.POMPAGE.PP11.STATE_Off OR NOT PRG_POMPAGE.POMPAGE.PS11.STATE_Ar OR NOT PRG_POMPAGE.POMPAGE.OP_Marche_Pompes.AR; 	(*Mise en puissance compresseur*)

(*timer*)
FM_state_chaud(clk:=EAU.STATE_Chaud);
TIMER_chaud.PT		:=	PRM_tps_att_chaud;
TIMER_chaud.IN		:=	EAU.STATE_Chaud; (*FM_state_chaud.Q;*)
TIMER_chaud();

(* Affectation du tableau d'état des lignes d'eau *)
WATER[0]	:= TRUE;
FOR I:=1 TO 5 DO
	WATER[I]		:=	(LIGNE_REF[I].STATE_Ok AND EAU.STATE_Froid AND CONF_eau_chaude) OR
						(LIGNE_REF[I].STATE_Ok AND NOT CONF_eau_chaude);
	STATE_AR[I]		:=	(LIGNE_REF[I].STATE_Ar AND EAU.STATE_Froid AND CONF_eau_chaude) OR
						((*LIGNE_REF[I].STATE_Ok AND*) EAU.STATE_Chaud AND TIMER_chaud.Q AND CONF_eau_chaude) OR
						(LIGNE_REF[I].STATE_Ar AND NOT CONF_eau_chaude);
END_FOR;

END_FUNCTION_BLOCK

// ---- POUs/Fonction/FONCTIONS SERVITUDES/BLOCK_LIGNE_REF.TcPOU
FUNCTION_BLOCK BLOCK_LIGNE_REF

(* Fonction de gestion d'une ligne d'eau simple (Vanne avec ou sans débitmètre à seuil*)

(****************historique des versions*****************************)
(* Version 1-0 - SP - VERSION INITIALE - 6844*)
(* Version 1-1 - AB - Compatible eau chaude / eau froide - 6970*)
(*Version 2-0 SP - ajout des paramètres de définition d'objet - SP - 7326 BA8 *)
(*************************************************************************)
VAR_INPUT

	RESET:				BOOL;
	MANUAL:				BOOL;			(* ~ (OPC : 1 : available for OPC-clients) *)
	IN_DExT:			BOOL;			(* ~ (OPC : 1 : available for OPC-clients) *)		(*débitmètre d'eau*)

	CO_On:				BOOL;													(*commande de marche*)

	I_Cond_need_Ref:			BOOL;													(*condition qui necessite le refroidissement*)
	I_inhibe_surv_ref:			BOOL;													(*Condition d'inhibition de la surveillance du débit*)
	I_Cond_ref_Ok:				BOOL;													(*Condition de validation du bon refroidissment (Temp, ...) *)

	VEx:						BLOCK_ACTUATOR2;										(*vanne d'eau simple*)

	DEF_Ref:				PRCDEF;												(*défaut de refroidissement*)
	DEF_Dex:				PRCDEF;												(*défaut de fonctionnement du débitmètre*)

END_VAR

VAR_INPUT PERSISTENT
	CONF_NO_DexT:			BOOL;													(*option pas de débitmètre*)
	CONF_TIM_OFF:			TIME;			(* ~ (OPC : 1 : available for OPC-clients) *)		(*temps entre la perte de la condition absolue de refroidissement
																					et la fermeture de la vanne d'eau*)
	CONF_No_Def_Dex:		BOOL;													(*pas de surveillance du défaut de fermeture de la vanne*)

	CONF_Eau_chaude:		BOOL;			(*ligne d'eau raccordée à un circuit eau chaude/froide*)

	(*Entité*)
	IsAssembly:		BOOL;			(*entité : assemblage*)
	IdXML:			STRING;			(*nom entité : identifiant pour recherche dans dico*)
	TagXML:			UINT;			(*nom entité : identifiant pour recherche dans dico*)
	IdParent:		STRING;			(*MNEMO de l'appelant*)
	MNEMO:			STRING;			(*MNEMO de l'entité*)
	MNEMO_Dex:		STRING;			(*MNEMO du débitmètre*)
END_VAR

VAR_OUTPUT
	STATE_Ok:				BOOL;			(* ~ (OPC : 1 : available for OPC-clients) *)		(*refroidissement ok*)
	STATE_Ar:				BOOL;			(* ~ (OPC : 1 : available for OPC-clients) *)		(*refroidissement à l'arrêt*)
	STATE_Nok:				BOOL;			(* ~ (OPC : 1 : available for OPC-clients) *)		(*refroidissement à l'arrêt*)
	STATE_DexT:				BOOL;			(* ~ (OPC : 1 : available for OPC-clients) *)		(*seuil débitmètre*)
END_VAR

VAR
	TIMER_OFF:				TON;
	VAR_Etape:				USINT;												(*Etape du grafcet de gestion de la servitudes*)
END_VAR

Def_Ref.IdXML		:=	'8';
Def_Ref.TagXML		:=	1;

DEF_Dex.IdXML		:=	'8';
DEF_Dex.TagXML		:=	2;

VEx.IdParent				:=	MNEMO;
VEx.IdXML					:=	'1';
VEx.TagXML					:=	1;
VEx.DEF_Off_auto.IdXML		:=	'3';
VEx.DEF_Off_auto.TagXML		:=	11;
VEx.DEF_Off_Imposs.IdXML	:=	'3';
VEx.DEF_Off_Imposs.TagXML	:=	9;
VEx.DEF_On_Imposs.IdXML		:=	'3';
VEx.DEF_On_Imposs.TagXML	:=	6;


(* initialisation du grafcet*)
IF 		VAR_etape = 0
		THEN
				VAR_etape.0 := TRUE;
(*repositionnement sur étape 0*)
ELSIF	MANUAL OR RESET
		THEN
				VAR_etape := 0;				(*RAZ grafcet*)
				VAR_etape.0:= TRUE;
(*étape 0-1*)
ELSIF 	VAR_etape.0
		AND CO_On
		THEN
				VAR_etape.1:= TRUE;
				VAR_etape.0:= FALSE;
(*étape 1-0*)
ELSIF 	VAR_etape.1
		AND NOT CO_on AND TIMER_OFF.Q
		THEN
				VAR_etape.0:= TRUE;
				VAR_etape.1:= FALSE;
END_IF;

(*Traitement en sortie*)
TIMER_OFF.PT	:=	CONF_TIM_OFF;
TIMER_OFF.IN	:=	VAR_Etape.1 AND NOT  I_Cond_need_Ref;
TIMER_OFF();

(*bit d'état*)
IF		((VAR_Etape.1 AND (IN_DExT OR CONF_NO_DExT) AND NOT MANUAL AND VEx.OUT_On)
		OR (MANUAL AND (IN_DExT OR CONF_NO_DExT)  AND VEx.OUT_On)) AND I_Cond_ref_Ok THEN
	STATE_Ok	:=	TRUE;
ELSIF	(NOT VAR_Etape.1AND NOT MANUAL)
		OR DEF_Ref.DEF
		OR (MANUAL AND NOT IN_DExT AND NOT CONF_NO_DExT AND VEx.OUT_On)
		OR NOT VEx.OUT_On
		OR NOT I_Cond_ref_Ok THEN
	STATE_Ok	:=	FALSE;
END_IF
STATE_Ar		:=	(VAR_Etape.0 AND NOT MANUAL) OR (MANUAL AND NOT VEx.OUT_ON) OR RESET;
STATE_NOk		:=	DEF_Dex.DEF OR DEF_Ref.DEF;
STATE_DexT		:=	(IN_DExT OR CONF_NO_DexT);

(*Pilotage de la vanne*)
VEx(
	RESET:=				RESET ,
	MANUAL:=				MANUAL ,
	CO_On:=					VAR_Etape.1,
	CONF_EN_On:= 			1,
	CONF_No_Safety_Auto:=	0,
	CONF_Tim_Valid_On:=		T#200ms,
	CONF_Tim_Valid_Off:= 	T#200ms);


(*Défaut de refroidissement*)
DEF_Ref.CONDITION		:=	VEx.OUT_On AND NOT IN_DExt AND NOT CONF_NO_DexT AND NOT RESET
							AND NOT I_Inhibe_Surv_Ref;
DEF_Ref();

(*Défaut débitmètre ou fermeture vanne*)
DEF_DEx.CONDITION		:=	NOT VEx.OUT_On AND IN_DExT AND NOT CONF_No_Def_Dex AND NOT RESET AND NOT CONF_NO_DexT;
DEF_DEx.DELAY			:= 	T#60s;
DEF_DEx();

END_FUNCTION_BLOCK

// ---- POUs/Fonction/FONCTIONS SERVITUDES/BLOCK_WREFCH1.TcPOU
FUNCTION_BLOCK BLOCK_WREFCH1

(* Fonction standard AC de gestion de bacsulement eau chaude eau froide *)

(****************historique des versions*****************************)

(* Version 1-0 - SP - VERSION INIITIALE*)
(*Version 2-0 - HG - Adaptation pour journal des évènements externe - 27/06/2011*)
(*ATTENTION !!! VERSION SPECIAL 9070 - GV - Ajout gestion niveau haut eau chaude pour éviter le débordement du réservoir eau chaude*)

(*************************************************************************)
VAR_INPUT
	I_PARAM_SYSTEM_OK:		BOOL;			(*paramétrage système ok*)

	RESET:					BOOL;
	MANUAL:					BOOL;			(* ~ (OPC : 1 : available for OPC-clients) *)
	CTRL_PLC:				BOOL;

	OP_CHAUD:				BLOCK_OPERATION;										(*Opération de mise en eau chaude*)
	OP_FROID:				BLOCK_OPERATION;										(*Operation de mise ne eau froide*)

	VEF_IN:					BLOCK_ACTUATOR2;										(*vanne eau froid amont*)
	VEF_OUT:				BLOCK_ACTUATOR2;										(*vanne eau froid aval*)
	VEC_IN:					BLOCK_ACTUATOR2;										(*Vanne eau chaude amont*)
	VEC_OUT:				BLOCK_ACTUATOR2;										(*Vanne eau froide aval*)

	IN_NIV:					BOOL;													(*Capteur niveau haut eau chaude*)
	DEF_Egal_Eau:			PRCDEF;												(*Défaut d'égalisation du niveau d'eau chaude vers eau froide*)

END_VAR

VAR_INPUT PERSISTENT
	CONF_Tim_Step:			TIME;						(*Temps entre chaque ouverture / fermeture de vanne*)

	(*Entité*)
	IsAssembly:		BOOL;			(*entité : assembly*)
	IdXML:			STRING;			(*nom entité : identifiant pour recherche dans dico*)
	TagXML:			UINT;			(*nom entité : identifiant pour recherche dans dico*)
	IdParent:		STRING;			(*MNEMO de l'appelant*)
	MNEMO:			STRING;			(*MNEMO de l'entité*)
END_VAR

VAR_OUTPUT
	STATE_Froid:			BOOL;						(* ~ (OPC : 1 : available for OPC-clients) *)
	STATE_Chaud:			BOOL;						(* ~ (OPC : 1 : available for OPC-clients) *)
END_VAR

VAR
	TIMER1:					TON;
	TIMER2:					TON;
	TIMER3:					TON;
	VAR_VEC_Out:			BOOL;
	VAR_VEC_In:				BOOL;
	VAR_VEF_Out:			BOOL;
	VAR_VEF_In:				BOOL;
END_VAR

PRL();
ACT_CHAUD();
ACT_FROID();
POST();

ACTION ACT_CHAUD:
(* OPERATION MISE EN EAU CHAUDE*)


(*initialisation de l'opération*)
OP_CHAUD(
	CTRL_PLC:= CTRL_PLC,
	RESET:= RESET,
	ENABLE_INT:=TRUE,
	MANUAL:= MANUAL,
	ON_AUTO_INT:=  FALSE,
	RESTART_ENABLE_IF_OK:= FALSE,
	N_STEP_OP_OK:= 11,
	N_STEP_OP_NOK:=0);

(*appel de l'action de préparation de l'opération*)
OP_CHAUD.PRL();


(*GRAFCET*)
(* initialisation du grafcet*)
IF 		OP_Chaud.ETAPE = 0 THEN
				OP_Chaud.Etape.0 := TRUE;
(*repositionnement sur étape 0*)
ELSIF	MANUAL OR RESET OR OP_Froid.Etape.1 THEN
				OP_Chaud.Etape := 0;			(*RAZ grafcet*)
				OP_Chaud.Etape.0:=TRUE;
(*étape 0-1*)
ELSIF 	OP_Chaud.ETAPE.0
		AND OP_Chaud.MARCHE_OP THEN
				OP_Chaud.Etape.1:=TRUE;
				OP_Chaud.Etape.0:=FALSE;
(*étape 1-2*)
ELSIF	OP_Chaud.ETAPE.1
		AND OP_FROID.Etape.0
		THEN
				OP_Chaud.Etape.2:=TRUE;
				OP_Chaud.Etape.1:=FALSE;
(*étape 2-3*)
ELSIF 	OP_Chaud.Etape.2
		AND timer1.Q THEN
				OP_Chaud.Etape.3:=TRUE;
				OP_Chaud.Etape.2:=FALSE;
(*étape 3-4*)
ELSIF	OP_Chaud.Etape.3
		AND timer2.Q	THEN
				OP_Chaud.Etape.4:=TRUE;
				OP_Chaud.Etape.3:=FALSE;
(*étape 4-5*)
ELSIF 	OP_Chaud.Etape.4
		AND Timer1.Q THEN
				OP_Chaud.Etape.5:=TRUE;
				OP_Chaud.Etape.4:=FALSE;
(*étape 5-11*)
ELSIF 	OP_Chaud.ETAPE.5
		AND TIMER2.Q AND NOT IN_NIV THEN
				OP_Chaud.Etape.11:=TRUE;
				OP_Chaud.Etape.5:=FALSE;
(*étape 5-6*)
ELSIF	OP_Chaud.Etape.5
		AND IN_NIV THEN
				OP_Chaud.Etape.6:=TRUE;
				OP_Chaud.Etape.5:=FALSE;
(*étape 6-7*)
ELSIF	OP_Chaud.Etape.6
		AND VEC_OUT.STATE_Off
		THEN
				OP_Chaud.Etape.7:=TRUE;
				OP_Chaud.Etape.6:=FALSE;
(*étape 7-8*)
ELSIF	OP_Chaud.Etape.7
		AND VEF_OUT.STATE_On THEN
				OP_Chaud.Etape.8:=TRUE;
				OP_Chaud.Etape.7:=FALSE;
(*étape 8-9*)
ELSIF	OP_Chaud.Etape.8
		AND Timer3.Q OR DEF_Egal_Eau.DEF
		THEN
				OP_Chaud.Etape.9:=TRUE;
				OP_Chaud.Etape.8:=FALSE;
(*étape 9-10*)
ELSIF	OP_Chaud.Etape.9
		AND VEF_OUT.STATE_Off
		THEN
				OP_Chaud.Etape.10:=TRUE;
				OP_Chaud.Etape.9:=FALSE;
(*étape 10-11*)
ELSIF	OP_Chaud.Etape.10
		AND VEC_OUT.STATE_On
		THEN
				OP_Chaud.Etape.11:=TRUE;
				OP_Chaud.Etape.10:=FALSE;
END_IF;

(*cloture du traitement de l'opération*)
OP_CHAUD.POST();
END_ACTION

ACTION ACT_FROID:
(* OPERATION MISE EN EAU FROIDE*)


(*initialisation de l'opération*)
OP_FROID(
	CTRL_PLC:= CTRL_PLC,
	RESET:= RESET,
	ENABLE_INT:=TRUE,
	MANUAL:= MANUAL,
	ON_AUTO_INT:=  FALSE,
	RESTART_ENABLE_IF_OK:= FALSE,
	N_STEP_OP_OK:= 6,
	N_STEP_OP_NOK:=0);

(*appel de l'action de préparation de l'opération*)
OP_FROID.PRL();


(*GRAFCET*)
(* initialisation du grafcet*)
IF 		OP_FROID.ETAPE = 0 THEN
				OP_FROID.Etape.0 := TRUE;
(*repositionnement sur étape 0*)
ELSIF	MANUAL OR RESET OR OP_Chaud.Etape.1 THEN
				OP_FROID.Etape := 0;			(*RAZ grafcet*)
				OP_FROID.Etape.0:=TRUE;
(*étape 0-1*)
ELSIF 	OP_FROID.ETAPE.0
		AND OP_FROID.MARCHE_OP THEN
				OP_FROID.Etape.1:=TRUE;
				OP_FROID.Etape.0:=FALSE;
(*étape 1-2*)
ELSIF	OP_FROID.ETAPE.1
		AND OP_Chaud.Etape.0
		THEN
				OP_FROID.Etape.2:=TRUE;
				OP_FROID.Etape.1:=FALSE;
(*étape 2-3*)
ELSIF 	OP_FROID.Etape.2
		AND timer1.Q THEN
				OP_FROID.Etape.3:=TRUE;
				OP_FROID.Etape.2:=FALSE;
(*étape 3-4*)
ELSIF	OP_FROID.Etape.3
		AND timer2.Q	THEN
				OP_FROID.Etape.4:=TRUE;
				OP_FROID.Etape.3:=FALSE;
(*étape 4-5*)
ELSIF 	OP_FROID.Etape.4
		AND Timer1.Q THEN
				OP_FROID.Etape.5:=TRUE;
				OP_FROID.Etape.4:=FALSE;
(*étape 5-6*)
ELSIF 	OP_FROID.ETAPE.5
		AND TIMER2.Q THEN
				OP_FROID.Etape.6:=TRUE;
				OP_FROID.Etape.5:=FALSE;
END_IF;

(*cloture du traitement de l'opération*)
OP_FROID.POST();
END_ACTION

ACTION POST:
(*Défaut d'égalisation des niveaux d'eau*)
DEF_Egal_Eau.CONDITION		:= OP_CHAUD.Etape.8;
DEF_Egal_Eau.DELAY			:= T#15s;
DEF_Egal_Eau();

(*Timer*)
Timer1.PT	:=	CONF_Tim_Step;
Timer2.PT	:=	CONF_Tim_Step;
Timer3.PT	:=	T#10s;			 (*Temps additionel Transfert eau chaude vers eau froide*)
Timer1.in :=	OP_CHAUD.Etape.2 OR OP_Chaud.Etape.4 OR OP_froid.Etape.2 OR OP_froid.Etape.4;
Timer2.in :=	OP_CHAUD.Etape.3 OR OP_Chaud.Etape.5 OR OP_froid.Etape.3 OR OP_froid.Etape.5;
Timer3.in :=	OP_CHAUD.Etape.8 AND NOT IN_NIV;
Timer1();
Timer2();
Timer3();


(*pilotage de vannes*)
IF OP_Chaud.Etape.4 OR OP_Chaud.Etape.10 THEN
	VAR_VEC_Out	:=	TRUE;
ELSIF (OP_Chaud.Etape.0 AND OP_froid.Etape.0) OR OP_froid.etape.3 OR OP_Chaud.Etape.6 THEN
	VAR_VEC_Out	:=	FALSE;
END_IF;
IF OP_Chaud.Etape.5 THEN
	VAR_VEC_In		:=	TRUE;
ELSIF (OP_Chaud.Etape.0 AND OP_froid.Etape.0) OR OP_froid.etape.2 THEN
	VAR_VEC_In		:=	FALSE;
END_IF;
IF OP_Froid.Etape.4 OR OP_Chaud.Etape.7 THEN
	VAR_VEF_Out	:=	TRUE;
ELSIF (OP_Chaud.Etape.0 AND OP_froid.Etape.0) OR OP_chaud.etape.3 OR OP_Chaud.Etape.9 THEN
	VAR_VEF_Out	:=	FALSE;
END_IF;
IF OP_Froid.Etape.5 THEN
	VAR_VEF_In		:=	TRUE;
ELSIF (OP_Chaud.Etape.0 AND OP_Froid.Etape.0) OR OP_Chaud.etape.2 THEN
	VAR_VEF_In		:=	FALSE;
END_IF;

(*etat*)
STATE_Froid := (NOT MANUAL AND OP_FROID.OK) OR (MANUAL AND VEF_IN.STATE_On AND VEF_OUT.STATE_On);
STATE_Chaud := (NOT MANUAL AND OP_CHAUD.OK) OR (MANUAL AND VEC_IN.STATE_On AND VEC_OUT.STATE_On);

(*Vannes*)
VEC_IN(
	I_PARAM_SYSTEM_OK:= I_PARAM_SYSTEM_OK,
	RESET:=RESET ,
	MANUAL:=MANUAL ,
	CO_On:=VAR_VEC_In,
	EN_On_INT:=(VEF_OUT.STATE_Off AND VEF_IN.STATE_Off) OR (VEC_IN.STATE_On AND VEC_OUT.STATE_Off),
	EN_Off_INT:= TRUE,
	CONF_EN_On:= 0,
	CONF_No_Safety_Auto:=0,
	CONF_Tim_Valid_On:=T#200ms,
	CONF_Tim_Valid_Off:= T#200ms);

VEC_OUT(
	I_PARAM_SYSTEM_OK:= I_PARAM_SYSTEM_OK,
	RESET:=RESET ,
	MANUAL:=MANUAL ,
	CO_On:=VAR_VEC_Out,
	EN_On_INT:=VEF_OUT.STATE_Off AND VEF_IN.STATE_Off,
	EN_Off_INT:= TRUE,
	CONF_EN_On:= 0,
	CONF_No_Safety_Auto:=0,
	CONF_Tim_Valid_On:=T#200ms,
	CONF_Tim_Valid_Off:= T#200ms);

VEF_IN(
	I_PARAM_SYSTEM_OK:= I_PARAM_SYSTEM_OK,
	RESET:=RESET ,
	MANUAL:=MANUAL ,
	CO_On:= VAR_VEF_In,
	EN_On_INT:=VEC_OUT.STATE_Off AND VEC_IN.STATE_Off,
	EN_Off_INT:= TRUE,
	CONF_EN_On:= 0,
	CONF_No_Safety_Auto:=0,
	CONF_Tim_Valid_On:=T#200ms,
	CONF_Tim_Valid_Off:= T#200ms);

VEF_OUT(
	I_PARAM_SYSTEM_OK:= I_PARAM_SYSTEM_OK,
	RESET:=RESET ,
	MANUAL:=MANUAL ,
	CO_On:= VAR_VEF_Out,
	EN_On_INT:=(VEC_OUT.STATE_Off AND VEC_IN.STATE_Off) OR (VEC_IN.STATE_On AND VEC_OUT.STATE_Off),
	EN_Off_INT:= TRUE,
	CONF_EN_On:= 0,
	CONF_No_Safety_Auto:=0,
	CONF_Tim_Valid_On:=T#200ms,
	CONF_Tim_Valid_Off:= T#200ms);
END_ACTION

ACTION PRL:
IdXML			:=	'6';
TagXML			:=	2;

OP_CHAUD.IdParent	:=	MNEMO;
OP_CHAUD.MNEMO		:=	CONCAT(MNEMO,'_CHAUD');
OP_CHAUD.IdXML		:=	'5';
OP_CHAUD.TagXML		:=	1;

OP_FROID.IdParent	:=	MNEMO;
OP_FROID.MNEMO		:=	CONCAT(MNEMO,'_FROID');
OP_FROID.IdXML		:=	'5';
OP_FROID.TagXML		:=	2;

VEF_IN.IdXML					:=	'1';
VEF_IN.TagXML					:=	1;
VEF_IN.IdParent					:=	MNEMO;
VEF_IN.DEF_On_Imposs.IdXML		:=	'3';
VEF_IN.DEF_On_Imposs.TagXML		:=	6;
VEF_IN.DEF_Off_Imposs.IdXML		:=	'3';
VEF_IN.DEF_Off_Imposs.TagXML	:=	9;
VEF_IN.DEF_Off_auto.IdXML		:=	'3';
VEF_IN.DEF_Off_auto.TagXML		:=	11;

VEF_OUT.IdXML					:=	'1';
VEF_OUT.TagXML					:=	1;
VEF_OUT.IdParent				:=	MNEMO;
VEF_OUT.DEF_On_Imposs.IdXML		:=	'3';
VEF_OUT.DEF_On_Imposs.TagXML	:=	6;
VEF_OUT.DEF_Off_Imposs.IdXML	:=	'3';
VEF_OUT.DEF_Off_Imposs.TagXML	:=	9;
VEF_OUT.DEF_Off_auto.IdXML		:=	'3';
VEF_OUT.DEF_Off_auto.TagXML		:=	11;

VEC_IN.IdXML					:=	'1';
VEC_IN.TagXML					:=	1;
VEC_IN.IdParent					:=	MNEMO;
VEC_IN.DEF_On_Imposs.IdXML		:=	'3';
VEC_IN.DEF_On_Imposs.TagXML		:=	6;
VEC_IN.DEF_Off_Imposs.IdXML		:=	'3';
VEC_IN.DEF_Off_Imposs.TagXML	:=	9;
VEC_IN.DEF_Off_auto.IdXML		:=	'3';
VEC_IN.DEF_Off_auto.TagXML		:=	11;

VEC_OUT.IdXML					:=	'1';
VEC_OUT.TagXML					:=	1;
VEC_OUT.IdParent				:=	MNEMO;
VEC_OUT.DEF_On_Imposs.IdXML		:=	'3';
VEC_OUT.DEF_On_Imposs.TagXML	:=	6;
VEC_OUT.DEF_Off_Imposs.IdXML	:=	'3';
VEC_OUT.DEF_Off_Imposs.TagXML	:=	9;
VEC_OUT.DEF_Off_auto.IdXML		:=	'3';
VEC_OUT.DEF_Off_auto.TagXML		:=	11;

DEF_Egal_Eau.IdXML				:= '8';
DEF_Egal_Eau.TagXML				:= 4;
END_ACTION

END_FUNCTION_BLOCK

// ---- POUs/Programme/BLOCK_PRG_GAZ.TcPOU
FUNCTION_BLOCK BLOCK_PRG_GAZ

(*****************************************************************)
(* 		Programme ligne de gaz
		PRG_GAZ_TYPE_9070

		Gestion jusqu'à 4 lignes de gaz MFC_MKS
		+ EV SIMPLE
		+ Gestion d'une ligne de gaz sans débimètre
		4 POINT D'INJECTION PAR EV SIMPLE	max.		      

		Affaire 9070 : 2 ligne de gaz + 1 sans débimètre, pas de vanne d'injection + regulation de pression gaz ligne 1 & 2

		Version 0 - GV - 05/01/2015                                     
		FAMILLE : DP/AC			      
*)
(******************************************************************)

VAR_INPUT

	LIGNE_GAZ:				ARRAY[0..4] OF BLOCK_LIGNE_GAZ;
	DG:						ARRAY[0..4] OF BLOCK_MFC_MKS_NoCoE;
	VGIN:					ARRAY[0..4] OF BLOCK_ACTUATOR2;
	REGULATION_GAZ_L1:		BLOCK_REGUL_PR_GAZ;				(*regulation sur ligne 1*)
	REGULATION_GAZ_L2:		BLOCK_REGUL_PR_GAZ;				(*regulation sur ligne 2*)

	PRM_SEL_VGIN:	ARRAY[0..4] OF BOOL;					(*I_STANDARD --- Selection des vannes d'injection de gaz *)
END_VAR

VAR_INPUT PERSISTENT
	CONF_LIGNE_GAZ:		ARRAY[0..4] OF BOOL;		(*I_STANDARD -- Indique la présence de la ligne gaz sur le systeme*)
	CONF_VGIN:			ARRAY[0..4] OF BOOL;		(*I_STANDARD -- indique la présence des vannes d'injection de gaz sur le systeme*)
	CONF_NAME_VGIN:		ARRAY[0..4] OF STRING;		(*I_STANDARD -- Nom des point d'injection - par ex: cathode 1 / enceinte ...*)

	(*Entité*)
	IsAssembly:		BOOL;			(*entité : ensemble*)
	IdXML:			STRING;			(*nom entité : identifiant pour recherche dans dico*)
	TagXML:			UINT;			(*nom entité : identifiant pour recherche dans dico*)
	IdParent:		STRING;			(*MNEMO de l'appelant*)
	MNEMO:			STRING;			(*MNEMO de l'entité*)
END_VAR

VAR_OUTPUT
	OUT_VG11	AT %Q*:	BOOL;
	OUT_VG12	AT %Q*:	BOOL;
	OUT_VG13	AT %Q*:	BOOL;
	OUT_VG14	AT %Q*:	BOOL;
	OUT_VO2		AT%Q*:	BOOL;
	OUT_VGIN1	AT %Q*:	BOOL;
	OUT_VGIN2	AT %Q*:	BOOL;
	OUT_VGIN3	AT %Q*:	BOOL;
	OUT_VGIN4	AT %Q*:	BOOL;

	STATE_Ar:			BOOL;		(*I_STANDARD -indique que les fonctions puissances sont à l'arrêt*)
	STATE_Def_IProc:	BOOL;		(*I_STANDARD -indique la présence d'un défaut entrainant l'arrêt du procédé*)
END_VAR

(* Paramètre statique *)
(*General*)
IdXML				:=	'3';
TagXML				:=	0;

LIGNE_GAZ[1].IdXML			:=	'3';
LIGNE_GAZ[1].TagXML			:=	1;
LIGNE_GAZ[2].IdXML			:=	'3';
LIGNE_GAZ[2].TagXML			:=	2;
LIGNE_GAZ[3].IdXML			:=	'3';
LIGNE_GAZ[3].TagXML			:=	3;
LIGNE_GAZ[4].IdXML			:=	'3';
LIGNE_GAZ[4].TagXML			:=	4;

(*Configuration du programme*)
CONF_LIGNE_GAZ[1]	:=	TRUE;
CONF_LIGNE_GAZ[2]	:=	TRUE;
CONF_LIGNE_GAZ[3]	:=	FALSE;
CONF_LIGNE_GAZ[4]	:=	FALSE;
CONF_VGIN[1]		:=	FALSE;
CONF_VGIN[2]		:=	FALSE;
CONF_VGIN[3]		:=	FALSE;
CONF_VGIN[4]		:=	FALSE;


(*VG11*)
LIGNE_GAZ[1].VGI.CONF_Tim_Valid_Off		:=	T#1S;
LIGNE_GAZ[1].VGI.CONF_Tim_Valid_On		:=	T#1S;
LIGNE_GAZ[1].VGI.MNEMO					:=	'VG11';
LIGNE_GAZ[1].VGI.CONF_EN_On				:=	0;
LIGNE_GAZ[1].VGI.CONF_No_Safety_Auto	:=	FALSE;
(*VG12*)
LIGNE_GAZ[2].VGI.CONF_Tim_Valid_Off		:=	T#1S;
LIGNE_GAZ[2].VGI.CONF_Tim_Valid_On		:=	T#1S;
LIGNE_GAZ[2].VGI.MNEMO					:=	'VG12';
LIGNE_GAZ[2].VGI.CONF_EN_On				:=	0;
LIGNE_GAZ[2].VGI.CONF_No_Safety_Auto	:=	FALSE;
(*VG13*)
LIGNE_GAZ[3].VGI.CONF_Tim_Valid_Off		:=	T#1S;
LIGNE_GAZ[3].VGI.CONF_Tim_Valid_On		:=	T#1S;
LIGNE_GAZ[3].VGI.MNEMO					:=	'VG13';
LIGNE_GAZ[3].VGI.CONF_EN_On				:=	0;
LIGNE_GAZ[3].VGI.CONF_No_Safety_Auto	:=	FALSE;
(*VG14*)
LIGNE_GAZ[4].VGI.CONF_Tim_Valid_Off		:=	T#1S;
LIGNE_GAZ[4].VGI.CONF_Tim_Valid_On		:=	T#1S;
LIGNE_GAZ[4].VGI.MNEMO					:=	'VG14';
LIGNE_GAZ[4].VGI.CONF_EN_On				:=	0;
LIGNE_GAZ[4].VGI.CONF_No_Safety_Auto	:=	FALSE;

(*VGIN1*)
VGIN[1].MNEMO							:=	'VGIN1';
VGIN[1].IdXML							:=	'7';
VGIN[1].TagXML							:=	2;
VGIN[1].DEF_Off_auto.IdXML				:=	'3';
VGIN[1].DEF_Off_auto.TagXML				:=	11;
VGIN[1].DEF_Off_Imposs.IdXML			:=	'3';
VGIN[1].DEF_Off_Imposs.TagXML			:=	9;
VGIN[1].DEF_On_Imposs.IdXML				:=	'3';
VGIN[1].DEF_On_Imposs.TagXML			:=	6;
VGIN[1].CONF_Tim_Valid_Off				:=	T#1s;
VGIN[1].CONF_Tim_Valid_On				:=	T#1s;
VGIN[1].CONF_EN_On						:=	0;
VGIN[1].CONF_No_Safety_Auto				:=	FALSE;
(*VGIN2*)
VGIN[2].MNEMO							:=	'VGIN2';
VGIN[2].IdXML							:=	'7';
VGIN[2].TagXML							:=	2;
VGIN[2].DEF_Off_auto.IdXML				:=	'3';
VGIN[2].DEF_Off_auto.TagXML				:=	11;
VGIN[2].DEF_Off_Imposs.IdXML			:=	'3';
VGIN[2].DEF_Off_Imposs.TagXML			:=	9;
VGIN[2].DEF_On_Imposs.IdXML				:=	'3';
VGIN[2].DEF_On_Imposs.TagXML			:=	6;
VGIN[2].CONF_Tim_Valid_Off				:=	T#1s;
VGIN[2].CONF_Tim_Valid_On				:=	T#1s;
VGIN[2].CONF_EN_On						:=	0;
VGIN[2].CONF_No_Safety_Auto				:=	FALSE;
(*VGIN3*)
VGIN[3].MNEMO							:=	'VGIN3';
VGIN[3].IdXML							:=	'7';
VGIN[3].TagXML							:=	2;
VGIN[3].DEF_Off_auto.IdXML				:=	'3';
VGIN[3].DEF_Off_auto.TagXML				:=	11;
VGIN[3].DEF_Off_Imposs.IdXML			:=	'3';
VGIN[3].DEF_Off_Imposs.TagXML			:=	9;
VGIN[3].DEF_On_Imposs.IdXML				:=	'3';
VGIN[3].DEF_On_Imposs.TagXML			:=	6;
VGIN[3].CONF_Tim_Valid_Off				:=	T#1s;
VGIN[3].CONF_Tim_Valid_On				:=	T#1s;
VGIN[3].CONF_EN_On						:=	0;
VGIN[3].CONF_No_Safety_Auto				:=	FALSE;
(*VGIN4*)
VGIN[4].MNEMO							:=	'VGIN4';
VGIN[4].IdXML							:=	'7';
VGIN[4].TagXML							:=	2;
VGIN[4].DEF_Off_auto.IdXML				:=	'3';
VGIN[4].DEF_Off_auto.TagXML				:=	11;
VGIN[4].DEF_Off_Imposs.IdXML			:=	'3';
VGIN[4].DEF_Off_Imposs.TagXML			:=	9;
VGIN[4].DEF_On_Imposs.IdXML				:=	'3';
VGIN[4].DEF_On_Imposs.TagXML			:=	6;
VGIN[4].CONF_Tim_Valid_Off				:=	T#1s;
VGIN[4].CONF_Tim_Valid_On				:=	T#1s;
VGIN[4].CONF_EN_On						:=	0;
VGIN[4].CONF_No_Safety_Auto				:=	FALSE;

(*compteurs des vannes d'injection - pas de vanne présente *)
VGIN[1].VAR_CPT.DISABLE := TRUE;
VGIN[2].VAR_CPT.DISABLE := TRUE;
VGIN[3].VAR_CPT.DISABLE := TRUE;
VGIN[4].VAR_CPT.DISABLE := TRUE;

(*Débimètres*)
DG[1].MNEMO				:=	'DG11';
DG[2].MNEMO				:=	'DG12';
DG[3].MNEMO				:=	'DG13';
DG[4].MNEMO				:=	'DG14';

(*Regulation de gaz*)
REGULATION_GAZ_L1.CONF_Flow_Init	:=	1;	(*1 sccm pour mise en gaz*)
REGULATION_GAZ_L1.IdXML				:=	'3';
REGULATION_GAZ_L1.TagXML			:=	21;

REGULATION_GAZ_L2.CONF_Flow_Init	:=	1;	(*1 sccm pour mise en gaz*)
REGULATION_GAZ_L2.IdXML				:=	'3';
REGULATION_GAZ_L2.TagXML			:=	22;

(*Gestion du mode de pilotage*)
IF (MACHINE.RQ_Ctrl_Ihm OR MACHINE.STATE_Manu) THEN
	REGULATION_GAZ_L1.CTRL_PLC	:=	FALSE;
	REGULATION_GAZ_L2.CTRL_PLC	:=	FALSE;
	LIGNE_GAZ[3].CTRL_PLC := FALSE;
	LIGNE_GAZ[4].CTRL_PLC := FALSE;
ELSIF (MACHINE.RQ_Ctrl_Plc AND NOT MACHINE.STATE_Manu) THEN
	REGULATION_GAZ_L1.CTRL_PLC	:=	TRUE;
	REGULATION_GAZ_L2.CTRL_PLC	:=	TRUE;
	LIGNE_GAZ[3].CTRL_PLC := TRUE;
	LIGNE_GAZ[4].CTRL_PLC := TRUE;
END_IF

IF (MACHINE.RQ_Ctrl_Ihm OR MACHINE.STATE_Manu) AND NOT REGULATION_GAZ_L1.RQ_Ctrl_Gaz THEN
	LIGNE_GAZ[1].CTRL_PLC := FALSE;
ELSIF (MACHINE.RQ_Ctrl_Plc AND NOT MACHINE.STATE_Manu) OR REGULATION_GAZ_L1.RQ_Ctrl_Gaz THEN
	LIGNE_GAZ[1].CTRL_PLC := TRUE;
END_IF

IF (MACHINE.RQ_Ctrl_Ihm OR MACHINE.STATE_Manu) AND NOT REGULATION_GAZ_L2.RQ_Ctrl_Gaz THEN
	LIGNE_GAZ[2].CTRL_PLC := FALSE;
ELSIF (MACHINE.RQ_Ctrl_Plc AND NOT MACHINE.STATE_Manu) OR REGULATION_GAZ_L2.RQ_Ctrl_Gaz THEN
	LIGNE_GAZ[2].CTRL_PLC := TRUE;
END_IF


(*Ligne Gaz 1*)
PRG_GAZ.LIGNE_GAZ[1].OP_MARCHE.ON_PLC := MAIN.STEP_EMPILEMENT.RQ_MARCHE_GAZ[1];

PRG_GAZ.LIGNE_GAZ[1].OP_ARRET.ON_PLC :=	INIT_MACHINE.RQ_STOP_GAZ 
										OR MAIN.STEP_EMPILEMENT.RQ_ARRET_GAZ[1]
										OR REGULATION_GAZ_L1.RQ_Arret_Gaz;

IF REGULATION_GAZ_L1.RQ_Marche_Gaz THEN
	LIGNE_GAZ[1].PRM_Flow := REGULATION_GAZ_L1.CONF_Flow_Init;
	LIGNE_GAZ[1].OP_MARCHE.ON_PLC := TRUE;
END_IF

PRG_GAZ.REGULATION_GAZ_L1.OP_MARCHE.ON_PLC:= MAIN.STEP_EMPILEMENT.RQ_MARCHE_REGUL_GAZ[1];

PRG_GAZ.REGULATION_GAZ_L1.OP_ARRET.ON_PLC:=	INIT_MACHINE.RQ_STOP_GAZ OR
											MAIN.STEP_EMPILEMENT.RQ_ARRET_REGUL_GAZ[1];

(*Ligne Gaz 2*)
PRG_GAZ.LIGNE_GAZ[2].OP_MARCHE.ON_PLC := MAIN.STEP_EMPILEMENT.RQ_MARCHE_GAZ[2];

PRG_GAZ.LIGNE_GAZ[2].OP_ARRET.ON_PLC :=	INIT_MACHINE.RQ_STOP_GAZ
										OR MAIN.STEP_EMPILEMENT.RQ_ARRET_GAZ[2]
										OR REGULATION_GAZ_L2.RQ_Arret_Gaz;

IF REGULATION_GAZ_L2.RQ_Marche_Gaz THEN
	LIGNE_GAZ[2].PRM_Flow := REGULATION_GAZ_L2.CONF_Flow_Init;
	LIGNE_GAZ[2].OP_MARCHE.ON_PLC := TRUE;
END_IF

PRG_GAZ.REGULATION_GAZ_L2.OP_MARCHE.ON_PLC:= MAIN.STEP_EMPILEMENT.RQ_MARCHE_REGUL_GAZ[2];

PRG_GAZ.REGULATION_GAZ_L2.OP_ARRET.ON_PLC:=	INIT_MACHINE.RQ_STOP_GAZ OR
											MAIN.STEP_EMPILEMENT.RQ_ARRET_REGUL_GAZ[2];

(*Ligne Gaz 3*)
PRG_GAZ.LIGNE_GAZ[3].OP_MARCHE.ON_PLC := MAIN.STEP_EFFLUVAGE.RQ_MARCHE_GAZ[1];

PRG_GAZ.LIGNE_GAZ[3].OP_ARRET.ON_PLC := INIT_MACHINE.RQ_STOP_GAZ
										   OR MAIN.STEP_EFFLUVAGE.RQ_ARRET_GAZ;
										   
(*Ligne Gaz 4*)
PRG_GAZ.LIGNE_GAZ[4].OP_MARCHE.ON_PLC := MAIN.STEP_EFFLUVAGE.RQ_MARCHE_GAZ[2];

PRG_GAZ.LIGNE_GAZ[4].OP_ARRET.ON_PLC := INIT_MACHINE.RQ_STOP_GAZ
										   OR MAIN.STEP_EFFLUVAGE.RQ_ARRET_GAZ;


(*Paramétre dynamique*)
LIGNE_GAZ[1].OP_MARCHE.ENABLE_EXT		:= TRUE;
LIGNE_GAZ[2].OP_MARCHE.ENABLE_EXT		:= TRUE;
LIGNE_GAZ[3].OP_MARCHE.ENABLE_EXT		:= TRUE;
LIGNE_GAZ[4].OP_MARCHE.ENABLE_EXT		:= TRUE;
LIGNE_GAZ[1].OP_ARRET.ENABLE_EXT		:= TRUE;
LIGNE_GAZ[2].OP_ARRET.ENABLE_EXT		:= TRUE;
LIGNE_GAZ[3].OP_ARRET.ENABLE_EXT		:= TRUE;
LIGNE_GAZ[4].OP_ARRET.ENABLE_EXT		:= TRUE;
LIGNE_GAZ[1].VGI.EN_Off_EXT				:= TRUE;
LIGNE_GAZ[2].VGI.EN_Off_EXT				:= TRUE;
LIGNE_GAZ[3].VGI.EN_Off_EXT				:= TRUE;
LIGNE_GAZ[4].VGI.EN_Off_EXT				:= TRUE;
LIGNE_GAZ[1].VGI.EN_On_EXT				:= TRUE;
LIGNE_GAZ[2].VGI.EN_On_EXT				:= TRUE;
LIGNE_GAZ[3].VGI.EN_On_EXT				:= TRUE;
LIGNE_GAZ[4].VGI.EN_On_EXT				:= TRUE;
REGULATION_GAZ_L1.OP_MARCHE.ENABLE_EXT := REGULATION_GAZ_L2.OP_ARRET.OK;
REGULATION_GAZ_L2.OP_MARCHE.ENABLE_EXT := REGULATION_GAZ_L1.OP_ARRET.OK;

VGIN[1].EN_Off_EXT				:=	TRUE;
VGIN[1].EN_ON_EXT				:=	TRUE;
VGIN[2].EN_Off_EXT				:=	TRUE;
VGIN[2].EN_ON_EXT				:=	TRUE;
VGIN[3].EN_Off_EXT				:=	TRUE;
VGIN[3].EN_ON_EXT				:=	TRUE;
VGIN[4].EN_Off_EXT				:=	TRUE;
VGIN[4].EN_ON_EXT				:=	TRUE;

IF REGULATION_GAZ_L1.OP_MARCHE.Etape.6
	OR REGULATION_GAZ_L1.OP_MARCHE.Etape.7
	OR REGULATION_GAZ_L1.OP_MARCHE.AR THEN	(*marche gaz dans debut régulation, ou marche gaz classique, la consigne reste celle de la ligne de gaz*)
		DG[1].PRM_Flow := LIGNE_GAZ[1].OUT_DG_PRM_FLOW;
ELSIF REGULATION_GAZ_L1.OP_MARCHE.Etape.8		(*dans le cas de la regulation, la consigne devient celle du PID*)
	OR REGULATION_GAZ_L1.OP_MARCHE.Etape.9
	OR REGULATION_GAZ_L1.OP_MARCHE.Etape.10
	OR REGULATION_GAZ_L1.OP_MARCHE.Etape.11
	OR REGULATION_GAZ_L1.OP_MARCHE.Etape.12 THEN
		DG[1].PRM_Flow	:=	MIN(REGULATION_GAZ_L1.CONTROLEUR_GAZ.STATE_Flow, DG[1].CONF_Util_Max_Flow);
END_IF

LIGNE_GAZ[1]
	(
	RESET:= 			MACHINE.STATE_Off,
	MANUAL:=			MACHINE.STATE_Manu,
	VAC:= 				PRG_POMPAGE.VAC,
	DOOR:=				PRG_POMPAGE.DOOR ,
	PRM_Disable_Surv:=	(VGIN[1].STATE_Off OR NOT CONF_VGIN[1])
      						AND (VGIN[2].STATE_Off OR NOT CONF_VGIN[2])
      						AND (VGIN[3].STATE_Off OR NOT CONF_VGIN[3])
      						AND (VGIN[4].STATE_Off OR NOT CONF_VGIN[4])
      						AND NOT (NOT CONF_VGIN[1] AND NOT CONF_VGIN[2] AND NOT CONF_VGIN[3] AND NOT CONF_VGIN[4])
						OR REGULATION_GAZ_L1.OP_MARCHE.EC,		(*inhibition surveillance débit gaz si régulation en cours*)
	IN_DG_PRM_FLOW:=	DG[1].PRM_Flow,
	O_SURV_DISABLE=>  DG[1].I_SURV_DISABLE,
	);

IF REGULATION_GAZ_L2.OP_MARCHE.Etape.6
	OR REGULATION_GAZ_L2.OP_MARCHE.Etape.7
	OR REGULATION_GAZ_L2.OP_MARCHE.AR THEN	(*marche gaz dans debut régulation, ou marche gaz classique, la consigne reste celle de la ligne de gaz*)
		DG[2].PRM_Flow := LIGNE_GAZ[2].OUT_DG_PRM_FLOW;
ELSIF REGULATION_GAZ_L2.OP_MARCHE.Etape.8		(*dans le cas de la regulation, la consigne devient celle du PID*)
	OR REGULATION_GAZ_L2.OP_MARCHE.Etape.9
	OR REGULATION_GAZ_L2.OP_MARCHE.Etape.10
	OR REGULATION_GAZ_L2.OP_MARCHE.Etape.11
	OR REGULATION_GAZ_L2.OP_MARCHE.Etape.12 THEN
		DG[2].PRM_Flow	:=	MIN(REGULATION_GAZ_L2.CONTROLEUR_GAZ.STATE_Flow, DG[2].CONF_Util_Max_Flow);
END_IF

LIGNE_GAZ[2]
	(
	RESET:= 			MACHINE.STATE_Off,
	MANUAL:=			MACHINE.STATE_Manu,
	VAC:= 				PRG_POMPAGE.VAC,
	DOOR:=				PRG_POMPAGE.DOOR ,
	PRM_Disable_Surv:=	(VGIN[1].STATE_Off OR NOT CONF_VGIN[1])
     						AND (VGIN[2].STATE_Off OR NOT CONF_VGIN[2])
      						AND (VGIN[3].STATE_Off OR NOT CONF_VGIN[3])
     						AND (VGIN[4].STATE_Off OR NOT CONF_VGIN[4])
     						AND NOT (NOT CONF_VGIN[1] AND NOT CONF_VGIN[2] AND NOT CONF_VGIN[3] AND NOT CONF_VGIN[4])
						OR REGULATION_GAZ_L2.OP_MARCHE.EC,		(*inhibition surveillance débit gaz si régulation en cours*)
	IN_DG_PRM_FLOW:=	DG[2].PRM_Flow,
	O_SURV_DISABLE=> DG[2].I_SURV_DISABLE,
	);

LIGNE_GAZ[3]
	(
	RESET:= 			MACHINE.STATE_Off,
	MANUAL:=			MACHINE.STATE_Manu,
	VAC:= 				PRG_POMPAGE.M11.STATE_Seuil[14],
	DOOR:=				PRG_POMPAGE.DOOR ,
	PRM_Disable_Surv:=	(VGIN[1].STATE_Off OR NOT CONF_VGIN[1])
     						AND (VGIN[2].STATE_Off OR NOT CONF_VGIN[2])
      						AND (VGIN[3].STATE_Off OR NOT CONF_VGIN[3])
     						AND (VGIN[4].STATE_Off OR NOT CONF_VGIN[4])
      						AND NOT (NOT CONF_VGIN[1] AND NOT CONF_VGIN[2] AND NOT CONF_VGIN[3] AND NOT CONF_VGIN[4]),
	IN_DG_PRM_FLOW:=	DG[3].PRM_Flow,
	O_SURV_DISABLE=> DG[3].I_SURV_DISABLE,
	);
	
LIGNE_GAZ[4](
	RESET:= 			MACHINE.STATE_Off,
	MANUAL:=			MACHINE.STATE_Manu,
	VAC:= 				PRG_POMPAGE.M11.STATE_Seuil[14],
	DOOR:=				PRG_POMPAGE.DOOR ,
	PRM_Disable_Surv:=	(VGIN[1].STATE_Off OR NOT CONF_VGIN[1])
      						AND (VGIN[2].STATE_Off OR NOT CONF_VGIN[2])
      						AND (VGIN[3].STATE_Off OR NOT CONF_VGIN[3])
      						AND (VGIN[4].STATE_Off OR NOT CONF_VGIN[4])
      						AND NOT (NOT CONF_VGIN[1] AND NOT CONF_VGIN[2] AND NOT CONF_VGIN[3] AND NOT CONF_VGIN[4]),
	IN_DG_PRM_FLOW:=	DG[4].PRM_Flow,
	O_SURV_DISABLE=> DG[4].I_SURV_DISABLE,
	);

VGIN[1](
	I_PARAM_SYSTEM_OK:= PARAM_SYSTEM_OK,
	RESET:= MACHINE.STATE_Off,
	MANUAL:= MACHINE.STATE_Manu,
	CO_On:= PRM_SEL_VGIN[1] AND (
			LIGNE_GAZ[1].OP_MARCHE.OK OR
			LIGNE_GAZ[2].OP_MARCHE.OK OR
			LIGNE_GAZ[3].OP_MARCHE.OK OR
			LIGNE_GAZ[4].OP_MARCHE.OK )
	);
VGIN[2](
	I_PARAM_SYSTEM_OK:= PARAM_SYSTEM_OK,
	RESET:= MACHINE.STATE_Off,
	MANUAL:= MACHINE.STATE_Manu,
	CO_On:= PRM_SEL_VGIN[2] AND (
			LIGNE_GAZ[1].OP_MARCHE.OK OR
			LIGNE_GAZ[2].OP_MARCHE.OK OR
			LIGNE_GAZ[3].OP_MARCHE.OK OR
			LIGNE_GAZ[4].OP_MARCHE.OK )
	);
VGIN[3](
	I_PARAM_SYSTEM_OK:= PARAM_SYSTEM_OK,
	RESET:= MACHINE.STATE_Off,
	MANUAL:= MACHINE.STATE_Manu,
	CO_On:= PRM_SEL_VGIN[3] AND (
			LIGNE_GAZ[1].OP_MARCHE.OK OR
			LIGNE_GAZ[2].OP_MARCHE.OK OR
			LIGNE_GAZ[3].OP_MARCHE.OK OR
			LIGNE_GAZ[4].OP_MARCHE.OK )
	);
VGIN[4](
	I_PARAM_SYSTEM_OK:= PARAM_SYSTEM_OK,
	RESET:= MACHINE.STATE_Off,
	MANUAL:= MACHINE.STATE_Manu,
	CO_On:= PRM_SEL_VGIN[4] AND (
			LIGNE_GAZ[1].OP_MARCHE.OK OR
			LIGNE_GAZ[2].OP_MARCHE.OK OR
			LIGNE_GAZ[3].OP_MARCHE.OK OR
			LIGNE_GAZ[4].OP_MARCHE.OK )
	);

DG[3].PRM_Flow	:=	LIGNE_GAZ[3].OUT_DG_PRM_FLOW;
DG[4].PRM_Flow	:=	LIGNE_GAZ[4].OUT_DG_PRM_FLOW;

DG[1](
	RESET:= MACHINE.STATE_Off,
	);
DG[2](
	RESET:= MACHINE.STATE_Off,
	);
DG[3](
	RESET:= MACHINE.STATE_Off,
	);
DG[4](
	RESET:= MACHINE.STATE_Off,
	);

